// /Chiller_1_Trip
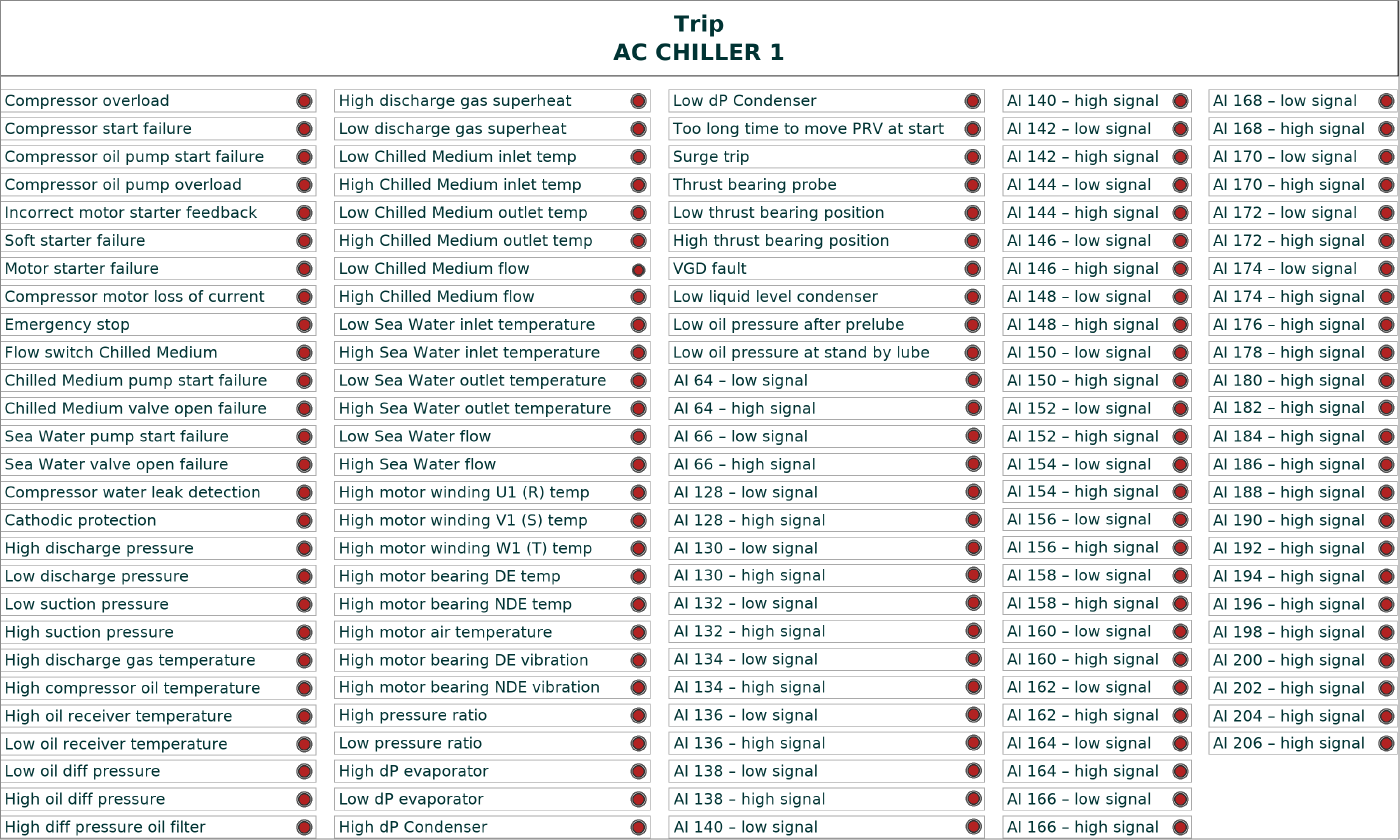
VISUALIZATION Chiller_1_Trip  // 1550x931
    Rectangle (0,0 1548x84)
    Label (318,7 912x70), "Trip AC CHILLER 1"
    Rectangle (0,99 350x25)
    Label (2,101 319x21), "Compressor overload"
    Lamp1 (326,102 22x20), variable: Chiller_1.T_Overload_compressor_motor, style: Lamp-Lamp1-Red
    Rectangle (0,130 350x25)
    Label (2,132 319x21), "Compressor start failure"
    Lamp1 (326,133 22x20), variable: Chiller_1.T_Starter_failure_trip, style: Lamp-Lamp1-Red
    Rectangle (0,161 350x25)
    Label (2,163 319x21), "Compressor oil pump start failure"
    Lamp1 (326,164 22x20), variable: Chiller_1.T_Oil_pump_running_failure, style: Lamp-Lamp1-Red
    Rectangle (0,192 350x25)
    Label (2,194 319x21), "Compressor oil pump overload"
    Lamp1 (326,195 22x20), variable: Chiller_1.T_Overload_oil_pump_motor, style: Lamp-Lamp1-Red
    Rectangle (0,223 350x25)
    Label (2,225 319x21), "Incorrect motor starter feedback"
    Lamp1 (326,226 22x20), variable: Chiller_1.T_Compressor_running_failure, style: Lamp-Lamp1-Red
    Rectangle (0,254 350x25)
    Label (2,256 319x21), "Soft starter failure"
    Lamp1 (326,257 22x20), variable: Chiller_1.T_Softstarter_failure, style: Lamp-Lamp1-Red
    Rectangle (0,285 350x25)
    Label (2,287 319x21), "Motor starter failure"
    Lamp1 (326,288 22x20), variable: Chiller_1.T_Motorstarter_failure, style: Lamp-Lamp1-Red
    Rectangle (0,316 350x25)
    Label (2,318 319x21), "Compressor motor loss of current"
    Lamp1 (326,319 22x20), variable: Chiller_1.T_Comp_motor_power_loss, style: Lamp-Lamp1-Red
    Rectangle (0,347 350x25)
    Label (2,349 319x21), "Emergency stop"
    Lamp1 (326,350 22x20), variable: Chiller_1.T_Emergency_stop, style: Lamp-Lamp1-Red
    Rectangle (0,378 350x25)
    Label (2,380 319x21), "Flow switch Chilled Medium"
    Lamp1 (326,381 22x20), variable: Chiller_1.T_Flow_switch_FT01, style: Lamp-Lamp1-Red
    Rectangle (0,409 350x25)
    Label (2,411 319x21), "Chilled Medium pump start failure"
    Lamp1 (326,412 22x20), variable: Chiller_1.T_Chilled_pump_run_failure, style: Lamp-Lamp1-Red
    Rectangle (0,440 350x25)
    Label (2,442 319x21), "Chilled Medium valve open failure"
    Lamp1 (326,443 22x20), variable: Chiller_1.T_CW_valveopen_failure, style: Lamp-Lamp1-Red
    Rectangle (0,471 350x25)
    Label (2,473 319x21), "Sea Water pump start failure"
    Lamp1 (326,474 22x20), variable: Chiller_1.T_Sea_water_pump_run_failure, style: Lamp-Lamp1-Red
    Rectangle (0,502 350x25)
    Label (2,504 319x21), "Sea Water valve open failure"
    Lamp1 (326,505 22x20), variable: Chiller_1.T_SW_valveopen_failure, style: Lamp-Lamp1-Red
    Rectangle (0,533 350x25)
    Label (2,535 319x21), "Compressor water leak detection"
    Lamp1 (326,536 22x20), variable: Chiller_1.T_Comp_motor_leak_detection, style: Lamp-Lamp1-Red
    Rectangle (0,564 350x25)
    Label (2,566 319x21), "Cathodic protection"
    Lamp1 (326,567 22x20), variable: Chiller_1.T_Cathodic_protect_sys_alarm, style: Lamp-Lamp1-Red
    Rectangle (0,595 350x25)
    Label (2,597 319x21), "High discharge pressure"
    Lamp1 (326,598 22x20), variable: Chiller_1.T_High_discharge_pressure, style: Lamp-Lamp1-Red
    Rectangle (0,626 350x25)
    Label (2,628 319x21), "Low discharge pressure"
    Lamp1 (326,629 22x20), variable: Chiller_1.T_Low_discharge_pressure, style: Lamp-Lamp1-Red
    Rectangle (0,688 350x25)
    Label (2,690 319x21), "High suction pressure"
    Lamp1 (326,691 22x20), variable: Chiller_1.T_High_suction_pressure, style: Lamp-Lamp1-Red
    Rectangle (0,657 350x25)
    Label (2,659 319x21), "Low suction pressure"
    Lamp1 (326,660 22x20), variable: Chiller_1.T_Low_suction_pressure, style: Lamp-Lamp1-Red
    Rectangle (0,719 350x25)
    Label (2,721 319x21), "High discharge gas temperature"
    Lamp1 (326,722 22x20), variable: Chiller_1.T_High_discharge_temp, style: Lamp-Lamp1-Red
    Rectangle (0,750 350x25)
    Label (2,752 319x21), "High compressor oil temperature"
    Lamp1 (326,753 22x20), variable: Chiller_1.T_High_temp_oil_inlet_comp, style: Lamp-Lamp1-Red
    Rectangle (0,781 350x25)
    Label (2,783 319x21), "High oil receiver temperature"
    Lamp1 (326,784 22x20), variable: Chiller_1.T_High_temp_oil_receiver, style: Lamp-Lamp1-Red
    Rectangle (370,749 350x25)
    Label (372,751 319x21), "High motor bearing NDE vibration"
    Lamp1 (696,752 22x20), variable: Chiller_1.T_High_comp_mot_NDE_bear_vib, style: Lamp-Lamp1-Red
    Rectangle (370,780 350x25)
    Label (372,782 319x21), "High pressure ratio"
    Lamp1 (696,783 22x20), variable: Chiller_1.T_High_press_ratio, style: Lamp-Lamp1-Red
    Rectangle (370,811 350x25)
    Label (372,813 319x21), "Low pressure ratio"
    Lamp1 (696,814 22x20), variable: Chiller_1.T_Low_press_ratio, style: Lamp-Lamp1-Red
    Rectangle (370,842 350x25)
    Label (372,844 319x21), "High dP evaporator"
    Lamp1 (696,845 22x20), variable: Chiller_1.T_High_CW_dP, style: Lamp-Lamp1-Red
    Rectangle (370,873 350x25)
    Label (372,875 319x21), "Low dP evaporator"
    Lamp1 (696,876 22x20), variable: Chiller_1.T_Low_CW_dP, style: Lamp-Lamp1-Red
    Rectangle (370,904 350x25)
    Label (372,906 319x21), "High dP Condenser"
    Lamp1 (696,907 22x20), variable: Chiller_1.T_High_SW_dP, style: Lamp-Lamp1-Red
    Rectangle (0,842 350x25)
    Label (2,844 319x21), "Low oil diff pressure"
    Lamp1 (326,845 22x20), variable: Chiller_1.T_Low_oil_diff_pressure, style: Lamp-Lamp1-Red
    Rectangle (0,873 350x25)
    Label (2,875 319x21), "High oil diff pressure"
    Lamp1 (326,876 22x20), variable: Chiller_1.T_High_diff_oil_pressure, style: Lamp-Lamp1-Red
    Rectangle (0,904 350x25)
    Label (2,906 319x21), "High diff pressure oil filter"
    Lamp1 (326,907 22x20), variable: Chiller_1.T_High_oil_filter_diff_press, style: Lamp-Lamp1-Red
    Rectangle (0,812 350x25)
    Label (2,814 319x21), "Low oil receiver temperature"
    Lamp1 (326,815 22x20), variable: Chiller_1.T_Low_temp_oil_receiver, style: Lamp-Lamp1-Red
    Rectangle (370,99 350x25)
    Label (372,101 319x21), "High discharge gas superheat"
    Lamp1 (696,102 22x20), variable: Chiller_1.T_High_disch_superheat, style: Lamp-Lamp1-Red
    Rectangle (370,130 350x25)
    Label (372,132 319x21), "Low discharge gas superheat"
    Lamp1 (696,133 22x20), variable: Chiller_1.T_Low_disch_superheat, style: Lamp-Lamp1-Red
    Rectangle (370,161 350x25)
    Label (372,163 319x21), "Low Chilled Medium inlet temp"
    Lamp1 (696,164 22x20), variable: Chiller_1.T_Low_CW_inlet_temp, style: Lamp-Lamp1-Red
    Rectangle (370,192 350x25)
    Label (372,194 319x21), "High Chilled Medium inlet temp"
    Lamp1 (696,195 22x20), variable: Chiller_1.T_High_CW_inlet_temp, style: Lamp-Lamp1-Red
    Rectangle (370,502 350x25)
    Label (372,504 319x21), "High Sea Water flow"
    Lamp1 (696,505 22x20), variable: Chiller_1.T_High_condenser_flow, style: Lamp-Lamp1-Red
    Rectangle (370,533 350x25)
    Label (372,535 319x21), "High motor winding U1 (R) temp"
    Lamp1 (696,536 22x20), variable: Chiller_1.T_High_motor_wind_temp_R, style: Lamp-Lamp1-Red
    Rectangle (370,564 350x25)
    Label (372,566 319x21), "High motor winding V1 (S) temp"
    Lamp1 (696,567 22x20), variable: Chiller_1.T_High_motor_wind_temp_S, style: Lamp-Lamp1-Red
    Rectangle (370,595 350x25)
    Label (372,597 319x21), "High motor winding W1 (T) temp"
    Lamp1 (696,598 22x20), variable: Chiller_1.T_High_motor_wind_temp_T, style: Lamp-Lamp1-Red
    Rectangle (370,626 350x25)
    Label (372,628 319x21), "High motor bearing DE temp"
    Lamp1 (696,629 22x20), variable: Chiller_1.T_High_comp_mot_DE_bear_temp, style: Lamp-Lamp1-Red
    Rectangle (370,657 350x25)
    Label (372,659 319x21), "High motor bearing NDE temp"
    Lamp1 (696,660 22x20), variable: Chiller_1.T_High_comp_mot_NDE_bear_temp, style: Lamp-Lamp1-Red
    Rectangle (370,688 350x25)
    Label (372,690 319x21), "High motor air temperature"
    Lamp1 (696,691 22x20), variable: Chiller_1.T_High_motor_air_temp, style: Lamp-Lamp1-Red
    Rectangle (370,223 350x25)
    Label (372,225 319x21), "Low Chilled Medium outlet temp"
    Lamp1 (696,226 22x20), variable: Chiller_1.T_Low_CW_outlet_temp, style: Lamp-Lamp1-Red
    Rectangle (370,254 350x25)
    Label (372,256 319x21), "High Chilled Medium outlet temp"
    Lamp1 (696,257 22x20), variable: Chiller_1.T_High_CW_outlet_temp, style: Lamp-Lamp1-Red
    Rectangle (370,285 350x25)
    Label (372,287 330x21), "Low Chilled Medium flow"
    Lamp1 (696,291 22x17), variable: Chiller_1.T_Low_chilled_medium_flow, style: Lamp-Lamp1-Red
    Rectangle (370,347 350x25)
    Label (372,349 319x21), "Low Sea Water inlet temperature"
    Lamp1 (696,350 22x20), variable: Chiller_1.T_Low_SW_inlet_temp, style: Lamp-Lamp1-Red
    Rectangle (370,378 350x25)
    Label (372,380 319x21), "High Sea Water inlet temperature"
    Lamp1 (696,381 22x20), variable: Chiller_1.T_High_SW_inlet_temp, style: Lamp-Lamp1-Red
    Rectangle (370,409 350x25)
    Label (372,411 319x21), "Low Sea Water outlet temperature"
    Lamp1 (696,412 22x20), variable: Chiller_1.T_Low_SW_outlet_temp, style: Lamp-Lamp1-Red
    Rectangle (370,440 350x25)
    Label (372,442 319x21), "High Sea Water outlet temperature"
    Lamp1 (696,443 22x20), variable: Chiller_1.T_High_SW_outlet_temp, style: Lamp-Lamp1-Red
    Rectangle (370,471 350x25)
    Label (372,473 319x21), "Low Sea Water flow"
    Lamp1 (696,474 22x20), variable: Chiller_1.T_Low_condenser_flow, style: Lamp-Lamp1-Red
    Rectangle (370,316 350x25)
    Label (372,318 319x21), "High Chilled Medium flow"
    Lamp1 (696,319 22x20), variable: Chiller_1.T_High_chilled_medium_flow, style: Lamp-Lamp1-Red
    Rectangle (370,719 350x25)
    Label (372,721 319x21), "High motor bearing DE vibration"
    Lamp1 (696,722 22x20), variable: Chiller_1.T_High_comp_mot_DE_bear_vib, style: Lamp-Lamp1-Red
    Rectangle (740,99 350x25)
    Label (742,101 319x21), "Low dP Condenser"
    Lamp1 (1066,102 22x20), variable: Chiller_1.T_Low_SW_dP, style: Lamp-Lamp1-Red
    Rectangle (740,130 350x25)
    Label (742,132 319x21), "Too long time to move PRV at start"
    Lamp1 (1066,133 22x20), variable: Chiller_1.T_Long_time_PRV, style: Lamp-Lamp1-Red
    Rectangle (740,161 350x25)
    Label (742,163 319x21), "Surge trip"
    Lamp1 (1066,164 22x20), variable: Chiller_1.T_Surge_detection, style: Lamp-Lamp1-Red
    Rectangle (740,378 350x25)
    Label (742,380 319x21), "Low oil pressure at stand by lube"
    Lamp1 (1066,381 22x20), variable: Chiller_1.T_Low_oilpress_standby, style: Lamp-Lamp1-Red
    Rectangle (740,192 350x25)
    Label (742,194 319x21), "Thrust bearing probe"
    Lamp1 (1066,195 22x20), variable: Chiller_1.T_Comp_thrust_bearing_position, style: Lamp-Lamp1-Red
    Rectangle (740,223 350x25)
    Label (742,225 319x21), "Low thrust bearing position"
    Lamp1 (1066,226 22x20), variable: Chiller_1.T_Comp_thrust_neg_move, style: Lamp-Lamp1-Red
    Rectangle (740,254 350x25)
    Label (742,256 319x21), "High thrust bearing position"
    Lamp1 (1066,257 22x20), variable: Chiller_1.T_Comp_thrust_pos_move, style: Lamp-Lamp1-Red
    Rectangle (740,285 350x25)
    Label (742,287 319x21), "VGD fault"
    Lamp1 (1066,288 22x20), variable: Chiller_1.T_VGD_fault, style: Lamp-Lamp1-Red
    Rectangle (740,316 350x25)
    Label (742,318 319x21), "Low liquid level condenser"
    Lamp1 (1066,319 22x20), variable: Chiller_1.T_Low_liquid_level, style: Lamp-Lamp1-Red
    Rectangle (740,347 350x25)
    Label (742,349 319x21), "Low oil pressure after prelube"
    Lamp1 (1066,350 22x20), variable: Chiller_1.T_Low_oilpress_prelube, style: Lamp-Lamp1-Red
    Rectangle (1110,316 209x25)
    Rectangle (1110,99 209x25)
    Rectangle (1110,130 209x25)
    Rectangle (1110,161 209x25)
    Rectangle (1110,192 209x25)
    Rectangle (1110,223 209x25)
    Rectangle (1110,254 209x25)
    Rectangle (1110,285 209x25)
    Rectangle (1110,347 209x25)
    Rectangle (1110,378 209x25)
    Rectangle (1110,409 209x25)
    Rectangle (1110,440 209x25)
    Rectangle (1110,471 209x25)
    Rectangle (1110,502 209x25)
    Lamp1 (1296,319 22x20), variable: Chiller_1.T_Sensor_low_signal_AI_148, style: Lamp-Lamp1-Red
    Lamp1 (1296,102 22x20), variable: Chiller_1.T_Sensor_high_signal_AI_140, style: Lamp-Lamp1-Red
    Lamp1 (1296,133 22x20), variable: Chiller_1.T_Sensor_low_signal_AI_142, style: Lamp-Lamp1-Red
    Lamp1 (1296,164 22x20), variable: Chiller_1.T_Sensor_high_signal_AI_142, style: Lamp-Lamp1-Red
    Lamp1 (1296,195 22x20), variable: Chiller_1.T_Sensor_low_signal_AI_144, style: Lamp-Lamp1-Red
    Lamp1 (1296,226 22x20), variable: Chiller_1.T_Sensor_high_signal_AI_144, style: Lamp-Lamp1-Red
    Lamp1 (1296,257 22x20), variable: Chiller_1.T_Sensor_low_signal_AI_146, style: Lamp-Lamp1-Red
    Lamp1 (1296,288 22x20), variable: Chiller_1.T_Sensor_high_signal_AI_146, style: Lamp-Lamp1-Red
    Lamp1 (1296,350 22x20), variable: Chiller_1.T_Sensor_high_signal_AI_148, style: Lamp-Lamp1-Red
    Lamp1 (1296,381 22x20), variable: Chiller_1.T_Sensor_low_signal_AI_150, style: Lamp-Lamp1-Red
    Lamp1 (1296,412 22x20), variable: Chiller_1.T_Sensor_high_signal_AI_150, style: Lamp-Lamp1-Red
    Lamp1 (1296,443 22x20), variable: Chiller_1.T_Sensor_low_signal_AI_152, style: Lamp-Lamp1-Red
    Lamp1 (1296,474 22x20), variable: Chiller_1.T_Sensor_high_signal_AI_152, style: Lamp-Lamp1-Red
    Label (1112,318 179x21), "AI 148 – low signal"
    Label (1112,101 179x21), "AI 140 – high signal"
    Label (1112,132 179x21), "AI 142 – low signal"
    Label (1112,163 179x21), "AI 142 – high signal"
    Label (1112,194 179x21), "AI 144 – low signal"
    Label (1112,225 179x21), "AI 144 – high signal"
    Label (1112,256 179x21), "AI 146 – low signal"
    Label (1112,287 179x21), "AI 146 – high signal"
    Label (1112,349 179x21), "AI 148 – high signal"
    Label (1112,380 179x21), "AI 150 – low signal"
    Label (1112,411 179x21), "AI 150 – high signal"
    Label (1112,442 179x21), "AI 152 – low signal"
    Label (1112,473 179x21), "AI 152 – high signal"
    Label (1112,504 179x21), "AI 154 – low signal"
    Lamp1 (1296,505 22x20), variable: Chiller_1.T_Sensor_low_signal_AI_154, style: Lamp-Lamp1-Red
    Rectangle (1110,532 209x25)
    Label (1112,534 179x21), "AI 154 – high signal"
    Lamp1 (1296,535 22x20), variable: Chiller_1.T_Sensor_high_signal_AI_154, style: Lamp-Lamp1-Red
    Rectangle (1110,563 209x25)
    Rectangle (1110,594 209x25)
    Rectangle (1110,625 209x25)
    Rectangle (1110,656 209x25)
    Rectangle (1110,687 209x25)
    Rectangle (1110,718 209x25)
    Rectangle (1110,749 209x25)
    Rectangle (1110,780 209x25)
    Rectangle (1110,811 209x25)
    Rectangle (1110,842 209x25)
    Rectangle (1110,873 209x25)
    Rectangle (1110,904 209x25)
    Lamp1 (1296,566 22x20), variable: Chiller_1.T_Sensor_low_signal_AI_156, style: Lamp-Lamp1-Red
    Lamp1 (1296,597 22x20), variable: Chiller_1.T_Sensor_high_signal_AI_156, style: Lamp-Lamp1-Red
    Lamp1 (1296,628 22x20), variable: Chiller_1.T_Sensor_low_signal_AI_158, style: Lamp-Lamp1-Red
    Lamp1 (1296,659 22x20), variable: Chiller_1.T_Sensor_high_signal_AI_158, style: Lamp-Lamp1-Red
    Lamp1 (1296,690 22x20), variable: Chiller_1.T_Sensor_low_signal_AI_160, style: Lamp-Lamp1-Red
    Lamp1 (1296,721 22x20), variable: Chiller_1.T_Sensor_high_signal_AI_160, style: Lamp-Lamp1-Red
    Lamp1 (1296,752 22x20), variable: Chiller_1.T_Sensor_low_signal_AI_162, style: Lamp-Lamp1-Red
    Lamp1 (1296,783 22x20), variable: Chiller_1.T_Sensor_high_signal_AI_162, style: Lamp-Lamp1-Red
    Lamp1 (1296,814 22x20), variable: Chiller_1.T_Sensor_low_signal_AI_164, style: Lamp-Lamp1-Red
    Lamp1 (1296,845 22x20), variable: Chiller_1.T_Sensor_high_signal_AI_164, style: Lamp-Lamp1-Red
    Lamp1 (1296,876 22x20), variable: Chiller_1.T_Sensor_low_signal_AI_166, style: Lamp-Lamp1-Red
    Lamp1 (1296,907 22x20), variable: Chiller_1.T_Sensor_high_signal_AI_166, style: Lamp-Lamp1-Red
    Label (1112,565 179x21), "AI 156 – low signal"
    Label (1112,596 179x21), "AI 156 – high signal"
    Label (1112,627 179x21), "AI 158 – low signal"
    Label (1112,658 179x21), "AI 158 – high signal"
    Label (1112,689 179x21), "AI 160 – low signal"
    Label (1112,720 179x21), "AI 160 – high signal"
    Label (1112,751 179x21), "AI 162 – low signal"
    Label (1112,782 179x21), "AI 162 – high signal"
    Label (1112,813 179x21), "AI 164 – low signal"
    Label (1112,844 179x21), "AI 164 – high signal"
    Label (1112,875 179x21), "AI 166 – low signal"
    Label (1112,906 179x21), "AI 166 – high signal"
    Rectangle (1338,223 209x25)
    Rectangle (1338,99 209x25)
    Rectangle (1338,130 209x25)
    Rectangle (1338,161 209x25)
    Rectangle (1338,192 209x25)
    Rectangle (1338,254 209x25)
    Rectangle (1338,285 209x25)
    Rectangle (1338,316 209x25)
    Rectangle (1338,347 209x25)
    Rectangle (1338,378 209x25)
    Rectangle (1338,409 209x25)
    Lamp1 (1524,226 22x20), variable: Chiller_1.T_Sensor_low_signal_AI_172, style: Lamp-Lamp1-Red
    Lamp1 (1524,102 22x20), variable: Chiller_1.T_Sensor_low_signal_AI_168, style: Lamp-Lamp1-Red
    Lamp1 (1524,133 22x20), variable: Chiller_1.T_Sensor_high_signal_AI_168, style: Lamp-Lamp1-Red
    Lamp1 (1524,164 22x20), variable: Chiller_1.T_Sensor_low_signal_AI_170, style: Lamp-Lamp1-Red
    Lamp1 (1524,195 22x20), variable: Chiller_1.T_Sensor_high_signal_AI_170, style: Lamp-Lamp1-Red
    Lamp1 (1524,257 22x20), variable: Chiller_1.T_Sensor_high_signal_AI_172, style: Lamp-Lamp1-Red
    Lamp1 (1524,288 22x20), variable: Chiller_1.T_Sensor_low_signal_AI_174, style: Lamp-Lamp1-Red
    Lamp1 (1524,319 22x20), variable: Chiller_1.T_Sensor_high_signal_AI_174, style: Lamp-Lamp1-Red
    Lamp1 (1524,350 22x20), variable: Chiller_1.T_Sensor_high_signal_AI_176, style: Lamp-Lamp1-Red
    Lamp1 (1524,381 22x20), variable: Chiller_1.T_Sensor_high_signal_AI_178, style: Lamp-Lamp1-Red
    Label (1340,225 179x21), "AI 172 – low signal"
    Label (1340,101 179x21), "AI 168 – low signal"
    Label (1340,132 179x21), "AI 168 – high signal"
    Label (1340,163 179x21), "AI 170 – low signal"
    Label (1340,194 179x21), "AI 170 – high signal"
    Label (1340,256 179x21), "AI 172 – high signal"
    Label (1340,287 179x21), "AI 174 – low signal"
    Label (1340,318 179x21), "AI 174 – high signal"
    Label (1340,349 179x21), "AI 176 – high signal"
    Label (1340,380 179x21), "AI 178 – high signal"
    Label (1340,411 179x21), "AI 180 – high signal"
    Lamp1 (1524,412 22x20), variable: Chiller_1.T_Sensor_high_signal_AI_180, style: Lamp-Lamp1-Red
    Rectangle (1338,439 209x25)
    Label (1340,441 179x21), "AI 182 – high signal"
    Lamp1 (1524,442 22x20), variable: Chiller_1.T_Sensor_high_signal_AI_182, style: Lamp-Lamp1-Red
    Rectangle (740,656 350x25)
    Rectangle (740,687 350x25)
    Rectangle (740,718 350x25)
    Rectangle (740,749 350x25)
    Rectangle (740,780 350x25)
    Rectangle (740,811 350x25)
    Rectangle (740,842 350x25)
    Rectangle (740,873 350x25)
    Rectangle (740,904 350x25)
    Label (743,658 299x21), "AI 132 – low signal"
    Label (743,689 299x21), "AI 132 – high signal"
    Label (743,720 299x21), "AI 134 – low signal"
    Label (743,751 299x21), "AI 134 – high signal"
    Label (743,782 299x21), "AI 136 – low signal"
    Label (743,813 299x21), "AI 136 – high signal"
    Label (743,844 299x21), "AI 138 – low signal"
    Label (743,875 299x21), "AI 138 – high signal"
    Label (743,906 299x21), "AI 140 – low signal"
    Rectangle (740,625 350x25)
    Rectangle (740,502 350x25)
    Rectangle (740,533 350x25)
    Rectangle (740,564 350x25)
    Rectangle (740,595 350x25)
    Rectangle (740,409 350x25)
    Rectangle (740,440 350x25)
    Rectangle (740,471 350x25)
    Label (743,504 298x21), "AI 66 – high signal"
    Label (743,535 298x21), "AI 128 – low signal"
    Label (743,566 298x21), "AI 128 – high signal"
    Label (743,597 298x21), "AI 130 – low signal"
    Label (743,411 298x21), "AI 64 – low signal"
    Label (743,442 298x21), "AI 64 – high signal"
    Label (743,473 298x21), "AI 66 – low signal"
    Label (743,627 350x21), "AI 130 – high signal"
    Lamp1 (1066,658 24x20), variable: Chiller_1.T_Sensor_low_signal_AI_132, style: Lamp-Lamp1-Red
    Lamp1 (1066,689 24x20), variable: Chiller_1.T_Sensor_high_signal_AI_132, style: Lamp-Lamp1-Red
    Lamp1 (1066,720 24x20), variable: Chiller_1.T_Sensor_low_signal_AI_134, style: Lamp-Lamp1-Red
    Lamp1 (1066,751 24x20), variable: Chiller_1.T_Sensor_high_signal_AI_134, style: Lamp-Lamp1-Red
    Lamp1 (1066,782 24x20), variable: Chiller_1.T_Sensor_low_signal_AI_136, style: Lamp-Lamp1-Red
    Lamp1 (1066,813 24x20), variable: Chiller_1.T_Sensor_high_signal_AI_136, style: Lamp-Lamp1-Red
    Lamp1 (1066,844 24x20), variable: Chiller_1.T_Sensor_low_signal_AI_138, style: Lamp-Lamp1-Red
    Lamp1 (1066,875 24x20), variable: Chiller_1.T_Sensor_high_signal_AI_138, style: Lamp-Lamp1-Red
    Lamp1 (1066,906 24x20), variable: Chiller_1.T_Sensor_low_signal_AI_140, style: Lamp-Lamp1-Red
    Lamp1 (1066,504 24x20), variable: Chiller_1.T_Sensor_high_signal_AI_66, style: Lamp-Lamp1-Red
    Lamp1 (1066,535 24x20), variable: Chiller_1.T_Sensor_low_signal_AI_128, style: Lamp-Lamp1-Red
    Lamp1 (1066,566 24x20), variable: Chiller_1.T_Sensor_high_signal_AI_128, style: Lamp-Lamp1-Red
    Lamp1 (1066,597 24x20), variable: Chiller_1.T_Sensor_low_signal_AI_130, style: Lamp-Lamp1-Red
    Lamp1 (1066,411 24x20), variable: Chiller_1.T_Sensor_low_signal_AI_64, style: Lamp-Lamp1-Red
    Lamp1 (1066,442 24x20), variable: Chiller_1.T_Sensor_high_signal_AI_64, style: Lamp-Lamp1-Red
    Lamp1 (1066,473 24x20), variable: Chiller_1.T_Sensor_low_signal_AI_66, style: Lamp-Lamp1-Red
    Lamp1 (1066,627 24x20), variable: Chiller_1.T_Sensor_high_signal_AI_130, style: Lamp-Lamp1-Red
    Rectangle (1338,595 209x25)
    Rectangle (1338,471 209x25)
    Rectangle (1338,502 209x25)
    Rectangle (1338,533 209x25)
    Rectangle (1338,564 209x25)
    Rectangle (1338,626 209x25)
    Rectangle (1338,657 209x25)
    Rectangle (1338,688 209x25)
    Rectangle (1338,719 209x25)
    Rectangle (1338,750 209x25)
    Rectangle (1338,781 209x25)
    Lamp1 (1524,598 22x20), variable: Chiller_1.T_Sensor_high_signal_AI_192, style: Lamp-Lamp1-Red
    Lamp1 (1524,474 22x20), variable: Chiller_1.T_Sensor_high_signal_AI_184, style: Lamp-Lamp1-Red
    Lamp1 (1524,505 22x20), variable: Chiller_1.T_Sensor_high_signal_AI_186, style: Lamp-Lamp1-Red
    Lamp1 (1524,536 22x20), variable: Chiller_1.T_Sensor_high_signal_AI_188, style: Lamp-Lamp1-Red
    Lamp1 (1524,567 22x20), variable: Chiller_1.T_Sensor_high_signal_AI_190, style: Lamp-Lamp1-Red
    Lamp1 (1524,629 22x20), variable: Chiller_1.T_Sensor_high_signal_AI_194, style: Lamp-Lamp1-Red
    Lamp1 (1524,660 22x20), variable: Chiller_1.T_Sensor_high_signal_AI_196, style: Lamp-Lamp1-Red
    Lamp1 (1524,691 22x20), variable: Chiller_1.T_Sensor_high_signal_AI_198, style: Lamp-Lamp1-Red
    Lamp1 (1524,722 22x20), variable: Chiller_1.T_Sensor_high_signal_AI_200, style: Lamp-Lamp1-Red
    Lamp1 (1524,753 22x20), variable: Chiller_1.T_Sensor_high_signal_AI_202, style: Lamp-Lamp1-Red
    Label (1340,597 179x21), "AI 192 – high signal"
    Label (1340,473 179x21), "AI 184 – high signal"
    Label (1340,504 179x21), "AI 186 – high signal"
    Label (1340,535 179x21), "AI 188 – high signal"
    Label (1340,566 179x21), "AI 190 – high signal"
    Label (1340,628 179x21), "AI 194 – high signal"
    Label (1340,659 179x21), "AI 196 – high signal"
    Label (1340,690 179x21), "AI 198 – high signal"
    Label (1340,721 179x21), "AI 200 – high signal"
    Label (1340,752 179x21), "AI 202 – high signal"
    Label (1340,783 179x21), "AI 204 – high signal"
    Lamp1 (1524,784 22x20), variable: Chiller_1.T_Sensor_high_signal_AI_204, style: Lamp-Lamp1-Red
    Rectangle (1338,811 209x25)
    Label (1340,813 179x21), "AI 206 – high signal"
    Lamp1 (1524,814 22x20), variable: Chiller_1.T_Sensor_high_signal_AI_206, style: Lamp-Lamp1-Red
END_VISUALIZATION

// /Chiller_1_Values
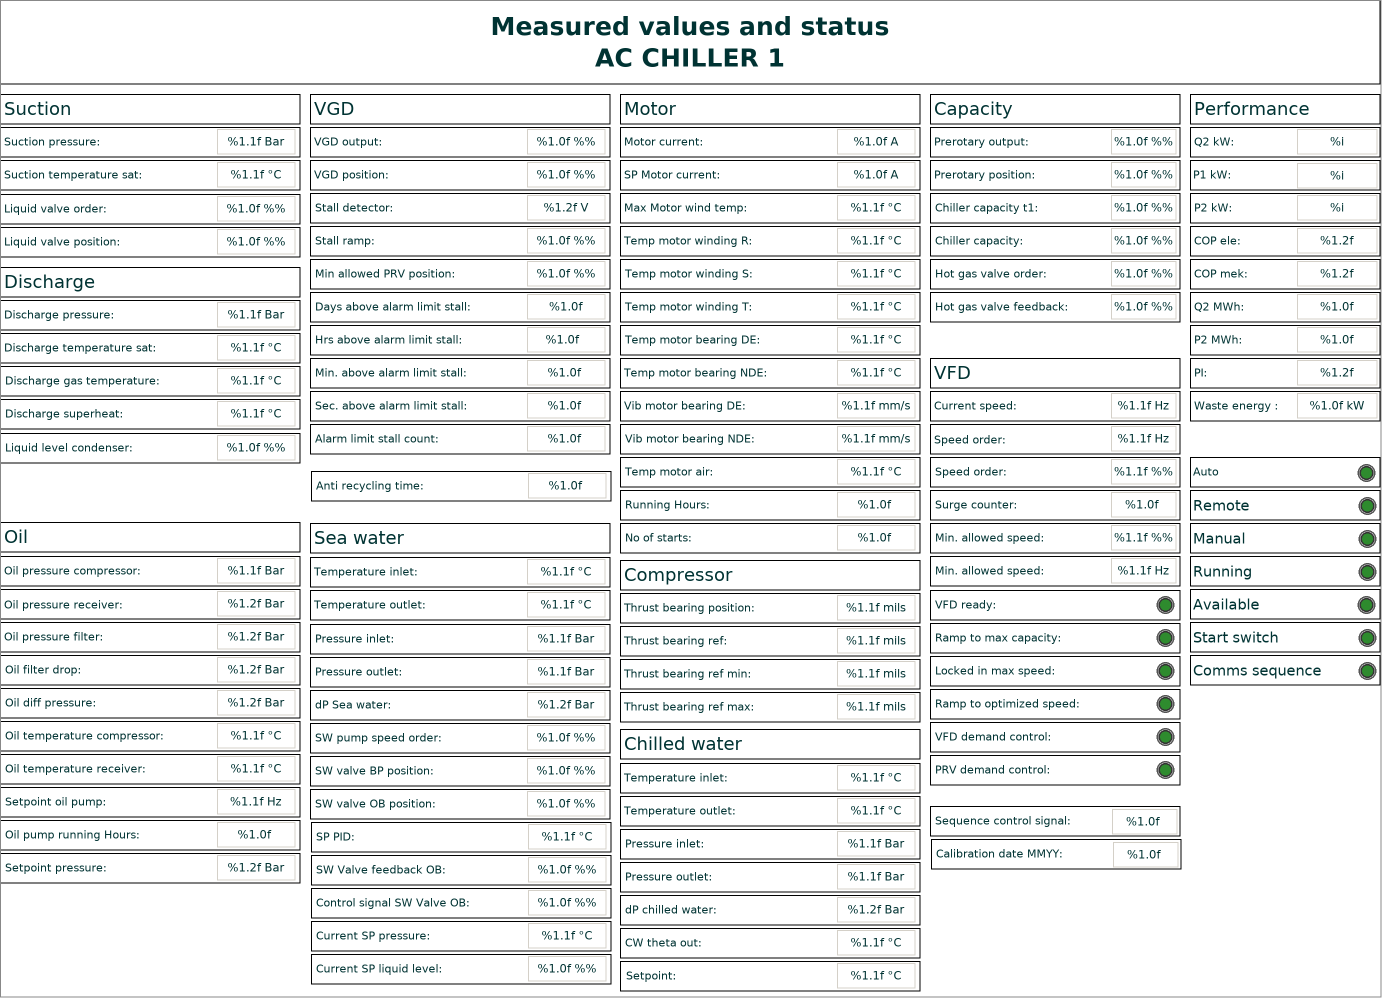
VISUALIZATION Chiller_1_Values  // 1382x998
    Rectangle (0,0 1380x84)
    Label (234,7 912x70), "Measured values and status AC CHILLER 1"
    Rectangle (0,94 300x30)
    Label (1,94 215x30), "Suction"
    Rectangle (0,127 300x30)
    Label (1,122 208x40), "Suction pressure:"
    Textfield (217,129 78x25), "%1.1f Bar", tooltip "Chiller_1.Press_suction_compr", text variable: Chiller_1.Press_suction_compr
        p4168582468: Chiller_1.Press_suction_compr
    Rectangle (0,160 300x30)
    Label (1,155 209x40), "Suction temperature sat:"
    Textfield (217,162 78x25), "%1.1f °C", tooltip "Chiller_1.Suction_saturated_temp", text variable: Chiller_1.Suction_saturated_temp
        p4168582468: Chiller_1.Suction_saturated_temp
    Rectangle (0,194 300x30)
    Label (1,189 211x40), "Liquid valve order:"
    Textfield (217,196 78x25), "%1.0f %%", tooltip "Chiller_1.Liquid_valve_output", text variable: Chiller_1.Liquid_valve_output
        p4168582468: Chiller_1.Liquid_valve_output
    Rectangle (0,227 300x30)
    Label (1,222 216x40), "Liquid valve position:"
    Textfield (217,229 78x25), "%1.0f %%", tooltip "Chiller_1.Feedback_liquid_valve", text variable: Chiller_1.Feedback_liquid_valve
        p4168582468: Chiller_1.Feedback_liquid_valve
    Rectangle (0,267 300x30)
    Label (1,267 194x30), "Discharge"
    Rectangle (0,300 300x30)
    Label (1,295 213x40), "Discharge pressure:"
    Textfield (217,302 78x25), "%1.1f Bar", tooltip "Chiller_1.Press_discharge_compr", text variable: Chiller_1.Press_discharge_compr
        p4168582468: Chiller_1.Press_discharge_compr
    Rectangle (0,333 300x30)
    Label (1,328 214x40), "Discharge temperature sat:"
    Textfield (217,335 78x25), "%1.1f °C", tooltip "Chiller_1.Discharge_saturated_temp", text variable: Chiller_1.Discharge_saturated_temp
        p4168582468: Chiller_1.Discharge_saturated_temp
    Rectangle (0,366 300x30)
    Label (2,361 213x40), "Discharge gas temperature:"
    Textfield (217,368 78x25), "%1.1f °C", tooltip "Chiller_1.Temp_discharge", text variable: Chiller_1.Temp_discharge
        p4168582468: Chiller_1.Temp_discharge
    Rectangle (0,433 300x30)
    Textfield (217,435 78x25), "%1.0f %%", tooltip "Chiller_1.Liquid_level_condenser", text variable: Chiller_1.Liquid_level_condenser
        p4168582468: Chiller_1.Liquid_level_condenser
    Rectangle (0,399 300x30)
    Label (2,394 212x40), "Discharge superheat:"
    Textfield (217,401 78x25), "%1.1f °C", tooltip "Chiller_1.Discharge_superheat", text variable: Chiller_1.Discharge_superheat
        p4168582468: Chiller_1.Discharge_superheat
    Rectangle (620,729 300x30)
    Label (621,729 194x30), "Chilled water"
    Rectangle (620,763 300x30)
    Label (621,758 204x40), "Temperature inlet:"
    Textfield (837,765 78x25), "%1.1f °C", tooltip "Chiller_1.Temp_chilled_medium_in", text variable: Chiller_1.Temp_chilled_medium_in
        p4168582468: Chiller_1.Temp_chilled_medium_in
    Rectangle (620,796 300x30)
    Label (621,791 209x40), "Temperature outlet:"
    Textfield (837,798 78x25), "%1.1f °C", tooltip "Chiller_1.Temp_chilled_medium_out", text variable: Chiller_1.Temp_chilled_medium_out
        p4168582468: Chiller_1.Temp_chilled_medium_out
    Rectangle (620,829 300x30)
    Label (622,824 206x40), "Pressure inlet:"
    Textfield (837,831 78x25), "%1.1f Bar", tooltip "Chiller_1.Press_chilled_medium_in", text variable: Chiller_1.Press_chilled_medium_in
        p4168582468: Chiller_1.Press_chilled_medium_in
    Rectangle (620,862 300x30)
    Label (622,857 208x40), "Pressure outlet:"
    Textfield (837,864 78x25), "%1.1f Bar", tooltip "Chiller_1.Press_chilled_medium_out", text variable: Chiller_1.Press_chilled_medium_out
        p4168582468: Chiller_1.Press_chilled_medium_out
    Rectangle (620,895 300x30)
    Label (622,890 207x40), "dP chilled water:"
    Textfield (837,897 78x25), "%1.2f Bar", tooltip "Chiller_1.dP_CW", text variable: Chiller_1.dP_CW
        p4168582468: Chiller_1.dP_CW
    Rectangle (620,928 300x30)
    Label (622,923 205x40), "CW theta out:"
    Textfield (837,930 78x25), "%1.1f °C", tooltip "Chiller_1.Theta_out", text variable: Chiller_1.Theta_out
        p4168582468: Chiller_1.Theta_out
    Rectangle (310,94 300x30)
    Label (311,94 194x30), "VGD"
    Rectangle (310,127 300x30)
    Label (311,122 209x40), "VGD output:"
    Textfield (527,129 78x25), "%1.0f %%", tooltip "Chiller_1.VGD_output", text variable: Chiller_1.VGD_output
        p4168582468: Chiller_1.VGD_output
    Rectangle (310,160 300x30)
    Label (311,155 204x40), "VGD position:"
    Textfield (527,162 78x25), "%1.0f %%", tooltip "Chiller_1.Feedback_VGD", text variable: Chiller_1.Feedback_VGD
        p4168582468: Chiller_1.Feedback_VGD
    Rectangle (310,193 300x30)
    Label (312,188 209x40), "Stall detector:"
    Textfield (527,195 78x25), "%1.2f V", tooltip "Chiller_1.Stall_detector", text variable: Chiller_1.Stall_detector
        p4168582468: Chiller_1.Stall_detector
    Rectangle (310,226 300x30)
    Label (312,221 178x40), "Stall ramp:"
    Textfield (527,228 78x25), "%1.0f %%", tooltip "Chiller_1.Stall_ramp", text variable: Chiller_1.Stall_ramp
        p4168582468: Chiller_1.Stall_ramp
    Rectangle (310,259 300x30)
    Label (312,254 216x40), "Min allowed PRV position:"
    Textfield (527,261 78x25), "%1.0f %%", tooltip "Chiller_1.Min_allowed_PRVposition", text variable: Chiller_1.Min_allowed_PRVposition
        p4168582468: Chiller_1.Min_allowed_PRVposition
    Rectangle (310,292 300x30)
    Label (312,287 216x40), "Days above alarm limit stall:"
    Textfield (527,294 78x25), "%1.0f", tooltip "Chiller_1.Days_above_stall_limit", text variable: Chiller_1.Days_above_stall_limit
        p4168582468: Chiller_1.Days_above_stall_limit
    Rectangle (310,325 300x30)
    Label (312,320 215x40), "Hrs above alarm limit stall:"
    Textfield (527,327 78x25), "%1.0f", tooltip "Chiller_1.Hrs_above_stall_limit", text variable: Chiller_1.Hrs_above_stall_limit
        p4168582468: Chiller_1.Hrs_above_stall_limit
    Rectangle (310,358 300x30)
    Label (312,353 218x40), "Min. above alarm limit stall:"
    Textfield (527,360 78x25), "%1.0f", tooltip "Chiller_1.Min_above_stall_limit", text variable: Chiller_1.Min_above_stall_limit
        p4168582468: Chiller_1.Min_above_stall_limit
    Rectangle (310,391 300x30)
    Label (312,386 214x40), "Sec. above alarm limit stall:"
    Textfield (527,393 78x25), "%1.0f", tooltip "Chiller_1.Sec_above_stall_limit", text variable: Chiller_1.Sec_above_stall_limit
        p4168582468: Chiller_1.Sec_above_stall_limit
    Rectangle (310,424 300x30)
    Label (312,419 216x40), "Alarm limit stall count:"
    Textfield (527,426 78x25), "%1.0f", tooltip "Chiller_1.Alarm_limit_stall_count", text variable: Chiller_1.Alarm_limit_stall_count
        p4168582468: Chiller_1.Alarm_limit_stall_count
    Rectangle (930,94 250x30)
    Label (931,94 162x30), "Capacity"
    Rectangle (930,127 250x30)
    Label (931,126 174x32), "Prerotary output:"
    Textfield (1111,129 65x25), "%1.0f %%", tooltip "Chiller_1.Prerotary_output", text variable: Chiller_1.Prerotary_output
        p4168582468: Chiller_1.Prerotary_output
    Rectangle (930,160 250x30)
    Label (931,159 173x32), "Prerotary position:"
    Textfield (1111,162 65x25), "%1.0f %%", tooltip "Chiller_1.Feedback_PRV", text variable: Chiller_1.Feedback_PRV
        p4168582468: Chiller_1.Feedback_PRV
    Rectangle (930,259 250x30)
    Label (932,258 177x32), "Hot gas valve order:"
    Textfield (1111,261 65x25), "%1.0f %%", tooltip "Chiller_1.Hot_gas_valve_output", text variable: Chiller_1.Hot_gas_valve_output
        p4168582468: Chiller_1.Hot_gas_valve_output
    Rectangle (930,292 250x30)
    Label (932,293 177x28), "Hot gas valve feedback:"
    Textfield (1111,294 65x25), "%1.0f %%", tooltip "Chiller_1.Feedback_HGV", text variable: Chiller_1.Feedback_HGV
        p4168582468: Chiller_1.Feedback_HGV
    Label (2,428 210x40), "Liquid level condenser:"
    Rectangle (310,523 300x30)
    Label (311,523 194x30), "Sea water"
    Rectangle (310,557 300x30)
    Label (311,552 211x40), "Temperature inlet:"
    Textfield (527,559 78x25), "%1.1f °C", tooltip "Chiller_1.Temp_water_inlet_cond", text variable: Chiller_1.Temp_water_inlet_cond
        p4168582468: Chiller_1.Temp_water_inlet_cond
    Rectangle (310,624 300x30)
    Label (312,619 210x40), "Pressure inlet:"
    Textfield (527,626 78x25), "%1.1f Bar", tooltip "Chiller_1.Press_water_cond_inlet", text variable: Chiller_1.Press_water_cond_inlet
        p4168582468: Chiller_1.Press_water_cond_inlet
    Rectangle (310,657 300x30)
    Label (312,652 210x40), "Pressure outlet:"
    Textfield (527,659 78x25), "%1.1f Bar", tooltip "Chiller_1.Press_water_cond_out", text variable: Chiller_1.Press_water_cond_out
        p4168582468: Chiller_1.Press_water_cond_out
    Rectangle (310,690 300x30)
    Label (312,685 210x40), "dP Sea water:"
    Textfield (527,692 78x25), "%1.2f Bar", tooltip "Chiller_1.dP_CW", text variable: Chiller_1.dP_SW
        p4168582468: Chiller_1.dP_SW
    Rectangle (310,723 300x30)
    Label (312,718 216x40), "SW pump speed order:"
    Textfield (527,725 78x25), "%1.0f %%", tooltip "Chiller_1.SW_pump_speed_order", text variable: Chiller_1.SW_pump_speed_order
        p4168582468: Chiller_1.SW_pump_speed_order
    Rectangle (310,756 300x30)
    Label (312,751 212x40), "SW valve BP position:"
    Textfield (527,758 78x25), "%1.0f %%", tooltip "Chiller_1.Order_SWW_bypass", text variable: Chiller_1.Order_SWW_bypass
        p4168582468: Chiller_1.Order_SWW_bypass
    Rectangle (310,789 300x30)
    Label (312,784 208x40), "SW valve OB position:"
    Textfield (527,791 78x25), "%1.0f %%", tooltip "Chiller_1.Order_SWW_overboard", text variable: Chiller_1.Order_SWW_overboard
        p4168582468: Chiller_1.Order_SWW_overboard
    Rectangle (310,590 300x30)
    Label (311,585 211x40), "Temperature outlet:"
    Textfield (527,592 78x25), "%1.1f °C", tooltip "Chiller_1.Temp_water_outlet_cond", text variable: Chiller_1.Temp_water_outlet_cond
        p4168582468: Chiller_1.Temp_water_outlet_cond
    Rectangle (0,522 300x30)
    Label (1,522 194x30), "Oil"
    Rectangle (0,556 300x30)
    Label (1,551 211x40), "Oil pressure compressor:"
    Textfield (217,558 78x25), "%1.1f Bar", tooltip "Chiller_1.Press_oil_compr", text variable: Chiller_1.Press_oil_compr
        p4168582468: Chiller_1.Press_oil_compr
    Rectangle (0,589 300x30)
    Label (1,585 210x40), "Oil pressure receiver:"
    Textfield (217,591 78x25), "%1.2f Bar", tooltip "Chiller_1.Press_oil_receiver", text variable: Chiller_1.Press_oil_receiver
        p4168582468: Chiller_1.Press_oil_receiver
    Rectangle (0,655 300x30)
    Label (2,650 209x40), "Oil filter drop:"
    Textfield (217,657 78x25), "%1.2f Bar", tooltip "Chiller_1.Oil_Filter_Drop", text variable: Chiller_1.Oil_Filter_Drop
        p4168582468: Chiller_1.Oil_Filter_Drop
    Rectangle (0,721 300x30)
    Label (2,716 218x40), "Oil temperature compressor:"
    Textfield (217,723 78x25), "%1.1f °C", tooltip "Chiller_1.Temp_oil_inlet_compr", text variable: Chiller_1.Temp_oil_inlet_compr
        p4168582468: Chiller_1.Temp_oil_inlet_compr
    Rectangle (0,754 300x30)
    Label (2,749 210x40), "Oil temperature receiver:"
    Textfield (217,756 78x25), "%1.1f °C", tooltip "Chiller_1.Oil_temp_receiver", text variable: Chiller_1.Oil_temp_receiver
        p4168582468: Chiller_1.Oil_temp_receiver
    Rectangle (0,688 300x30)
    Label (2,683 211x40), "Oil diff pressure:"
    Textfield (217,690 78x25), "%1.2f Bar", tooltip "Chiller_1.Oil_diff_pressure", text variable: Chiller_1.Oil_diff_pressure
        p4168582468: Chiller_1.Oil_diff_pressure
    Rectangle (0,787 300x30)
    Label (2,782 212x40), "Setpoint oil pump:"
    Textfield (217,789 78x25), "%1.1f Hz", tooltip "Chiller_1.Setpoint_conv_oil_pump", text variable: Chiller_1.Setpoint_conv_oil_pump
        p4168582468: Chiller_1.Setpoint_conv_oil_pump
    Rectangle (0,820 300x30)
    Label (2,815 206x40), "Oil pump running Hours:"
    Textfield (217,822 78x25), "%1.0f", tooltip "Chiller_1.Oil_pump_running_hours", text variable: Chiller_1.Oil_pump_running_hours
        p4168582468: Chiller_1.Oil_pump_running_hours
    Rectangle (0,622 300x30)
    Label (1,617 210x40), "Oil pressure filter:"
    Textfield (217,624 78x25), "%1.2f Bar", tooltip "Chiller_1.Oil_pressure_before_filter", text variable: Chiller_1.Oil_pressure_before_filter
        p4168582468: Chiller_1.Oil_pressure_before_filter
    Rectangle (620,560 300x30)
    Label (621,560 194x30), "Compressor"
    Rectangle (620,593 300x30)
    Label (621,592 216x32), "Thrust bearing position:"
    Textfield (837,595 78x25), "%1.1f mils", tooltip "Chiller_1.Thrust_bearing_position", text variable: Chiller_1.Thrust_bearing_position
        p4168582468: Chiller_1.Thrust_bearing_position
    Rectangle (620,659 300x30)
    Label (621,658 208x32), "Thrust bearing ref min:"
    Textfield (837,661 78x25), "%1.1f mils", tooltip "Chiller_1.Thrust_bearing_ref_min", text variable: Chiller_1.Thrust_bearing_ref_min
        p4168582468: Chiller_1.Thrust_bearing_ref_min
    Rectangle (1190,226 190x30)
    Label (1191,228 112x26), "COP ele:"
    Textfield (1297,228 80x25), "%1.2f", tooltip "Chiller_1.COP_chiller_ele", text variable: Chiller_1.COP_chiller_ele
        p4168582468: Chiller_1.COP_chiller_ele
    Rectangle (1190,94 190x30)
    Label (1191,94 123x30), "Performance"
    Rectangle (1190,127 190x30)
    Label (1191,126 112x32), "Q2 kW:"
    Textfield (1297,129 80x25), "%i", tooltip "Chiller_1.Chiller_capacity_kW", text variable: Chiller_1.Chiller_capacity_kW
        p4168582468: Chiller_1.Chiller_capacity_kW
    Rectangle (1190,193 190x30)
    Label (1191,194 112x28), "P2 kW:"
    Textfield (1297,195 80x25), "%i", tooltip "Chiller_1.P2_mot_1_kW", text variable: Chiller_1.P2_mot_1_kW
        p4168582468: Chiller_1.P2_mot_1_kW
    Rectangle (1190,160 190x30)
    Textfield (1297,163 80x25), "%i", tooltip "Chiller_1.P1_motor_kW", text variable: Chiller_1.P1_motor_kW
        p4168582468: Chiller_1.P1_motor_kW
    Label (1190,159 112x32), "P1 kW:"
    Rectangle (1190,457 190x30)
    Lamp1 (1355,463 23x20), tooltip "Chiller_1.Unit_auto", variable: Chiller_1.Unit_auto, style: Lamp-Lamp1-Green
    Label (1190,459 112x26), "Auto"
    Rectangle (1190,490 190x30)
    Rectangle (1190,523 190x30)
    Rectangle (1190,556 190x30)
    Rectangle (1190,589 190x30)
    Rectangle (1190,622 190x30)
    Rectangle (1190,655 190x30)
    Label (1190,495 105x21), "Remote"
    Lamp1 (1356,496 23x20), tooltip "Chiller_1.Unit_remote", variable: Chiller_1.Unit_remote, style: Lamp-Lamp1-Green
    Label (1190,528 105x21), "Manual"
    Lamp1 (1356,529 23x20), tooltip "Chiller_1.Unit_manual", variable: Chiller_1.Unit_manual, style: Lamp-Lamp1-Green
    Label (1190,561 105x21), "Running"
    Lamp1 (1356,562 23x20), tooltip "Chiller_1.Unit_running", variable: Chiller_1.Unit_running, style: Lamp-Lamp1-Green
    Label (1190,594 105x21), "Available"
    Lamp1 (1355,595 23x20), tooltip "Chiller_1.Unit_avabiable", variable: Chiller_1.Unit_available, style: Lamp-Lamp1-Green
    Label (1190,627 130x21), "Start switch"
    Lamp1 (1356,628 23x20), tooltip "Chiller_1.Unit_start_switch", variable: Chiller_1.Unit_start_switch, style: Lamp-Lamp1-Green
    Lamp1 (1356,661 23x20), tooltip "Sequence.A_Comms_chiller_1", variable: not.Sequence.A_Comms_chiller_1, style: Lamp-Lamp1-Green
    Label (1190,660 148x21), "Comms sequence"
    Rectangle (1190,292 190x30)
    Label (1191,293 112x28), "Q2 MWh:"
    Textfield (1297,294 80x25), "%1.0f", tooltip "Chiller_1.Q2_chillerMWh", text variable: Chiller_1.Q2_chillerMWh
        p4168582468: Chiller_1.Q2_chillerMWh
    Rectangle (930,358 250x30)
    Label (931,358 162x30), "VFD"
    Rectangle (930,391 250x30)
    Label (931,390 173x32), "Current speed:"
    Textfield (1111,393 65x25), "%1.1f Hz", tooltip "Chiller_1.Speed_feedback_VFD", text variable: Chiller_1.Speed_feedback_VFD
        p4168582468: Chiller_1.Speed_feedback_VFD
    Rectangle (930,424 250x30)
    Label (931,420 167x40), "Speed order:"
    Textfield (1111,426 65x25), "%1.1f Hz", tooltip "Chiller_1.Order_VFD_Hz", text variable: Chiller_1.Order_VFD_Hz
        p4168582468: Chiller_1.Order_VFD_Hz
    Rectangle (930,457 250x30)
    Label (932,455 171x34), "Speed order:"
    Textfield (1111,459 65x25), "%1.1f %%", tooltip "Chiller_1.Order_VFD_perc", text variable: Chiller_1.Order_VFD_perc
        p4168582468: Chiller_1.Order_VFD_perc
    Rectangle (930,490 250x30)
    Label (932,492 170x26), "Surge counter:"
    Textfield (1111,492 65x25), "%1.0f", tooltip "Chiller_1.Surge_counter_VFD", text variable: Chiller_1.Surge_counter_VFD
        p4168582468: Chiller_1.Surge_counter_VFD
    Rectangle (930,523 250x30)
    Label (932,522 176x32), "Min. allowed speed:"
    Textfield (1111,525 65x25), "%1.1f %%", tooltip "Chiller_1.Opt_speed_VFD_perc", text variable: Chiller_1.Opt_speed_VFD_perc
        p4168582468: Chiller_1.Opt_speed_VFD_perc
    Rectangle (930,556 250x30)
    Label (932,554 177x34), "Min. allowed speed:"
    Textfield (1111,558 65x25), "%1.1f Hz", tooltip "Chiller_1.Opt_speed_VFD_Hz", text variable: Chiller_1.Opt_speed_VFD_Hz
        p4168582468: Chiller_1.Opt_speed_VFD_Hz
    Rectangle (930,193 250x30)
    Label (932,192 174x32), "Chiller capacity t1:"
    Textfield (1111,195 65x25), "%1.0f %%", tooltip "Chiller_1.Chiller_capacity_t1", text variable: Chiller_1.Chiller_capacity_t1
        p4168582468: Chiller_1.Chiller_capacity_t1
    Rectangle (620,94 300x30)
    Label (621,94 194x30), "Motor"
    Rectangle (620,127 300x30)
    Label (621,122 209x40), "Motor current:"
    Textfield (837,129 78x25), "%1.0f A", tooltip "Chiller_1.Motor_current", text variable: Chiller_1.Motor_current
        p4168582468: Chiller_1.Motor_current
    Rectangle (620,226 300x30)
    Label (621,221 210x40), "Temp motor winding R:"
    Textfield (837,228 78x25), "%1.1f °C", tooltip "Chiller_1.Temp_motor_wind_R", text variable: Chiller_1.Temp_motor_wind_R
        p4168582468: Chiller_1.Temp_motor_wind_R
    Rectangle (620,259 300x30)
    Label (622,254 204x40), "Temp motor winding S:"
    Textfield (837,261 78x25), "%1.1f °C", tooltip "Chiller_1.Temp_motor_wind_S", text variable: Chiller_1.Temp_motor_wind_S
        p4168582468: Chiller_1.Temp_motor_wind_S
    Rectangle (620,292 300x30)
    Label (622,287 206x40), "Temp motor winding T:"
    Textfield (837,294 78x25), "%1.1f °C", tooltip "Chiller_1.Temp_motor_wind_T", text variable: Chiller_1.Temp_motor_wind_T
        p4168582468: Chiller_1.Temp_motor_wind_T
    Rectangle (620,325 300x30)
    Label (622,320 216x40), "Temp motor bearing DE:"
    Textfield (837,327 78x25), "%1.1f °C", tooltip "Chiller_1.Temp_motor_bearing_DE", text variable: Chiller_1.Temp_motor_bearing_DE
        p4168582468: Chiller_1.Temp_motor_bearing_DE
    Rectangle (620,358 300x30)
    Label (621,353 218x40), "Temp motor bearing NDE:"
    Textfield (837,360 78x25), "%1.1f °C", tooltip "Chiller_1.Temp_motor_bearing_NDE", text variable: Chiller_1.Temp_motor_bearing_NDE
        p4168582468: Chiller_1.Temp_motor_bearing_NDE
    Rectangle (620,391 300x30)
    Label (621,386 215x40), "Vib motor bearing DE:"
    Textfield (837,393 78x25), "%1.1f mm/s", tooltip "Chiller_1.Vibration_compressor_DE", text variable: Chiller_1.Vibration_compressor_DE
        p4168582468: Chiller_1.Vibration_compressor_DE
    Rectangle (620,424 300x30)
    Label (622,419 215x40), "Vib motor bearing NDE:"
    Textfield (837,426 78x25), "%1.1f mm/s", tooltip "Chiller_1.Vibration_compressor_NDE", text variable: Chiller_1.Vibration_compressor_NDE
        p4168582468: Chiller_1.Vibration_compressor_NDE
    Rectangle (620,457 300x30)
    Label (622,452 210x40), "Temp motor air:"
    Textfield (837,459 78x25), "%1.1f °C", tooltip "Chiller_1.Temp_motor_air", text variable: Chiller_1.Temp_motor_air
        p4168582468: Chiller_1.Temp_motor_air
    Rectangle (620,490 300x30)
    Label (622,485 204x40), "Running Hours:"
    Textfield (837,492 78x25), "%1.0f", tooltip "Chiller_1.Running_hours_compressormotor", text variable: Chiller_1.Running_hours_compressormotor
        p4168582468: Chiller_1.Running_hours_compressormotor
    Rectangle (620,523 300x30)
    Label (622,518 207x40), "No of starts:"
    Textfield (837,525 78x25), "%1.0f", tooltip "Chiller_1.Number_of_starts", text variable: Chiller_1.Number_of_starts
        p4168582468: Chiller_1.Number_of_starts
    Rectangle (930,590 250x30)
    Label (932,588 177x34), "VFD ready:"
    Lamp1 (1154,595 23x20), tooltip "Chiller_1.VFD_ready", variable: Chiller_1.VFD_ready, style: Lamp-Lamp1-Green
    Rectangle (930,623 250x30)
    Label (932,621 209x34), "Ramp to max capacity:"
    Lamp1 (1154,628 23x20), tooltip "Chiller_1.VFD_ramp_100_perc", variable: Chiller_1.VFD_ramp_100_perc, style: Lamp-Lamp1-Green
    Rectangle (930,656 250x30)
    Label (932,654 209x34), "Locked in max speed:"
    Lamp1 (1154,661 23x20), tooltip "Chiller_1.VFD_locked_100_perc", variable: Chiller_1.VFD_locked_100_perc, style: Lamp-Lamp1-Green
    Rectangle (930,689 250x30)
    Label (932,687 209x34), "Ramp to optimized speed:"
    Lamp1 (1154,694 23x20), tooltip "Chiller_1.VFD_ramp_d_PRVcontrol", variable: Chiller_1.VFD_ramp_d_PRVcontrol, style: Lamp-Lamp1-Green
    Rectangle (930,722 250x30)
    Label (932,720 209x34), "VFD demand control:"
    Lamp1 (1154,727 23x20), tooltip "Chiller_1.VFD_control", variable: Chiller_1.VFD_control, style: Lamp-Lamp1-Green
    Rectangle (930,755 250x30)
    Label (932,753 209x34), "PRV demand control:"
    Lamp1 (1154,760 23x20), tooltip "Chiller_1.PRV_control", variable: Chiller_1.PRV_control, style: Lamp-Lamp1-Green
    Rectangle (620,961 300x30)
    Label (623,956 205x40), "Setpoint:"
    Textfield (837,963 78x25), "%1.1f °C", tooltip "Chiller_1.SP_CW_controller", text variable: Chiller_1.SP_CW_controller
        p4168582468: Chiller_1.SP_CW_controller
    Rectangle (311,822 300x30)
    Label (313,817 208x40), "SP PID:"
    Textfield (528,824 78x25), "%1.1f °C", tooltip "Chiller_1.SP_PID_seawater", text variable: Chiller_1.SP_PID_seawater
        p4168582468: Chiller_1.SP_PID_seawater
    Rectangle (1190,259 190x30)
    Label (1191,261 112x26), "COP mek:"
    Textfield (1297,261 80x25), "%1.2f", tooltip "Chiller_1.COP_chiller_mech", text variable: Chiller_1.COP_chiller_mech
        p4168582468: Chiller_1.COP_chiller_mech
    Rectangle (620,692 300x30)
    Label (621,691 208x32), "Thrust bearing ref max:"
    Textfield (837,694 78x25), "%1.1f mils", tooltip "Chiller_1.Thrust_bearing_ref_max", text variable: Chiller_1.Thrust_bearing_ref_max
        p4168582468: Chiller_1.Thrust_bearing_ref_max
    Rectangle (620,160 300x30)
    Label (621,155 209x40), "SP Motor current:"
    Textfield (837,162 78x25), "%1.0f A", tooltip "Chiller_1.SP_MC_controller", text variable: Chiller_1.SP_MC_controller
        p4168582468: Chiller_1.SP_MC_controller
    Rectangle (620,626 300x30)
    Label (621,625 216x32), "Thrust bearing ref:"
    Textfield (837,628 78x25), "%1.1f mils", tooltip "Chiller_1.Thrust_bearing_ref", text variable: Chiller_1.Thrust_bearing_ref
        p4168582468: Chiller_1.Thrust_bearing_ref
    Rectangle (311,471 300x30)
    Label (313,466 216x40), "Anti recycling time:"
    Textfield (528,473 78x25), "%1.0f", tooltip "Chiller_1.Anti_recycle_time", text variable: Chiller_1.Anti_recycle_time
        p4168582468: Chiller_1.Anti_recycle_time
    Rectangle (0,853 300x30)
    Label (2,848 211x40), "Setpoint pressure:"
    Textfield (217,855 78x25), "%1.2f Bar", tooltip "Chiller_1.SP_oil_pressure", text variable: Chiller_1.SP_oil_pressure
        p4168582468: Chiller_1.SP_oil_pressure
    Rectangle (311,855 300x30)
    Label (313,850 208x40), "SW Valve feedback OB:"
    Textfield (528,857 78x25), "%1.0f %%", tooltip "Chiller_1.Feedback_seawater_valve_overboard", text variable: Chiller_1.Feedback_seawater_valve_overboard
        p4168582468: Chiller_1.Feedback_seawater_valve_overboard
    Rectangle (620,193 300x30)
    Label (621,188 210x40), "Max Motor wind temp:"
    Textfield (837,195 78x25), "%1.1f °C", tooltip "Chiller_1.Max_motor_wind_temp", text variable: Chiller_1.Max_motor_wind_temp
        p4168582468: Chiller_1.Max_motor_wind_temp
    Rectangle (311,888 300x30)
    Label (313,883 208x40), "Control signal SW Valve OB:"
    Textfield (528,890 78x25), "%1.0f %%", tooltip "Chiller_1.Feedback_seawater_valve_overboard", text variable: Chiller_1.Feedback_seawater_valve_overboard
        p4168582468: Chiller_1.Feedback_seawater_valve_overboard
    Rectangle (311,921 300x30)
    Label (313,916 208x40), "Current SP pressure:"
    Textfield (528,923 78x25), "%1.1f °C", tooltip "Chiller_1.SP_PID_seawater", text variable: Chiller_1.SP_cond_press
        p4168582468: Chiller_1.SP_PID_seawater
    Rectangle (311,954 300x30)
    Label (313,949 208x40), "Current SP liquid level:"
    Textfield (528,956 78x25), "%1.0f %%", tooltip "Chiller_1.SP_PID_Level", text variable: Chiller_1.SP_PID_Level
        p4168582468: Chiller_1.SP_PID_Level
    Rectangle (930,806 250x30)
    Label (932,804 183x34), "Sequence control signal:"
    Rectangle (1190,358 190x30)
    Label (1191,360 112x26), "PI:"
    Textfield (1297,360 80x25), "%1.2f", tooltip "Chiller_1.PI_chiller", text variable: Chiller_1.PI_chiller
        p4168582468: Chiller_1.PI_chiller
    Rectangle (1190,391 190x30)
    Label (1191,393 112x26), "Waste energy :"
    Textfield (1297,393 80x25), "%1.0f kW", tooltip "Chiller_1.Wasted_energy_kW", text variable: Chiller_1.Wasted_energy_kW
        p4168582468: Chiller_1.Wasted_energy_kW
    Rectangle (1190,325 190x30)
    Label (1191,327 112x26), "P2 MWh:"
    Textfield (1297,327 80x25), "%1.0f", tooltip "Chiller_1.Chiller_P2_MWh", text variable: Chiller_1.Chiller_P2_MWh
        p4168582468: Chiller_1.Chiller_P2_MWh
    Textfield (1112,809 65x25), "%1.0f", tooltip "Chiller_1.Control_signal_unit_d", text variable: Chiller_1.Control_signal_unit_d
        p4168582468: Chiller_1.Control_signal_unit_d
    Rectangle (931,839 250x30)
    Label (933,837 183x34), "Calibration date MMYY:"
    Textfield (1113,842 65x25), "%1.0f", tooltip "Chiller_1.Cal_date_MMYY", text variable: Chiller_1.Cal_date_MMYY
        p4168582468: Chiller_1.Cal_date_MMYY
    Rectangle (930,226 250x30)
    Label (932,225 174x32), "Chiller capacity:"
    Textfield (1111,228 65x25), "%1.0f %%", tooltip "Chiller_1.Chiller_capacity", text variable: Chiller_1.Chiller_capacity
        p4168582468: Chiller_1.Chiller_capacity
END_VISUALIZATION

// /Chiller_1_VFD
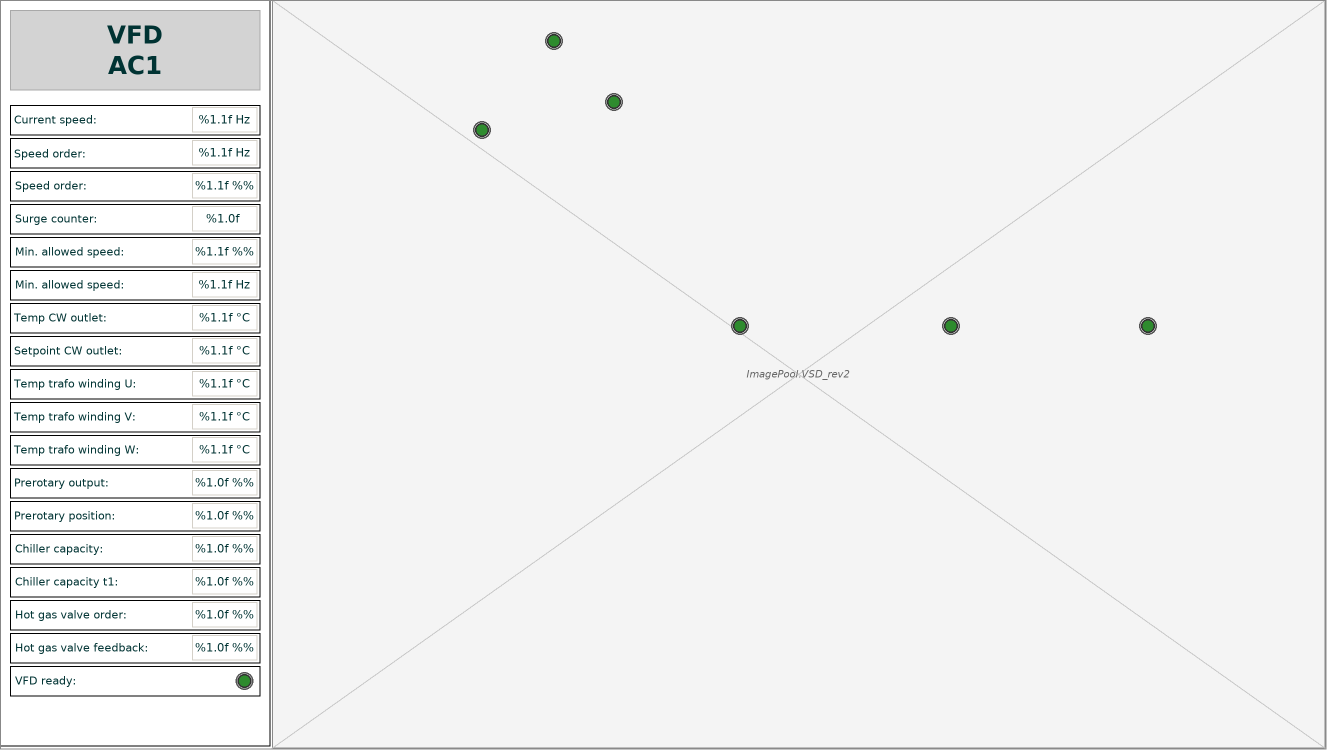
VISUALIZATION Chiller_1_VFD  // 1327x750
    Image (272,0 1053x748), image: ImagePool.VSD_rev2
    Rectangle (0,0 270x746)
    Lamp1 (469,120 26x20), variable: Chiller_1.VFD_ramp_100_perc, style: Lamp-Lamp1-Green
    Lamp1 (541,31 26x20), variable: Chiller_1.VFD_locked_100_perc, style: Lamp-Lamp1-Green
    Lamp1 (601,92 26x20), variable: Chiller_1.VFD_ramp_d_PRVcontrol, style: Lamp-Lamp1-Green
    Lamp1 (727,316 26x20), variable: Chiller_1.PRV_control, style: Lamp-Lamp1-Green
    Lamp1 (938,316 26x20), variable: Chiller_1.VFD_control, style: Lamp-Lamp1-Green
    Lamp1 (1135,316 26x20), variable: Chiller_1.PRV_control, style: Lamp-Lamp1-Green
    Textfield (10,10 250x80), "VFD AC1", text index: Sequence.Seq_cap_order_C3
    Rectangle (10,666 250x30)
    Label (12,664 177x34), "VFD ready:"
    Lamp1 (233,671 23x20), tooltip "Chiller_1.VFD_ready", variable: Chiller_1.VFD_ready, style: Lamp-Lamp1-Green
    Rectangle (10,105 250x30)
    Label (11,104 173x32), "Current speed:"
    Textfield (192,107 65x25), "%1.1f Hz", tooltip "Chiller_1.Speed_feedback_VFD", text variable: Chiller_1.Speed_feedback_VFD
        p4168582468: Chiller_1.Speed_feedback_VFD
    Rectangle (10,138 250x30)
    Label (11,134 167x40), "Speed order:"
    Textfield (192,140 65x25), "%1.1f Hz", tooltip "Chiller_1.Order_VFD_Hz", text variable: Chiller_1.Order_VFD_Hz
        p4168582468: Chiller_1.Order_VFD_Hz
    Rectangle (10,171 250x30)
    Label (12,169 171x34), "Speed order:"
    Textfield (192,173 65x25), "%1.1f %%", tooltip "Chiller_1.Order_VFD_perc", text variable: Chiller_1.Order_VFD_perc
        p4168582468: Chiller_1.Order_VFD_perc
    Rectangle (10,204 250x30)
    Label (12,206 170x26), "Surge counter:"
    Textfield (192,206 65x25), "%1.0f", tooltip "Chiller_1.Surge_counter_VFD", text variable: Chiller_1.Surge_counter_VFD
        p4168582468: Chiller_1.Surge_counter_VFD
    Rectangle (10,237 250x30)
    Label (12,236 176x32), "Min. allowed speed:"
    Textfield (192,239 65x25), "%1.1f %%", tooltip "Chiller_1.Opt_speed_VFD_perc", text variable: Chiller_1.Opt_speed_VFD_perc
        p4168582468: Chiller_1.Opt_speed_VFD_perc
    Rectangle (10,270 250x30)
    Label (12,268 177x34), "Min. allowed speed:"
    Textfield (192,272 65x25), "%1.1f Hz", tooltip "Chiller_1.Opt_speed_VFD_Hz", text variable: Chiller_1.Opt_speed_VFD_Hz
        p4168582468: Chiller_1.Opt_speed_VFD_Hz
    Rectangle (10,303 250x30)
    Label (11,305 169x26), "Temp CW outlet:"
    Textfield (192,305 65x25), "%1.1f °C", tooltip "Chiller_1.Temp_chilled_medium_out", text variable: Chiller_1.Temp_chilled_medium_out
        p4168582468: Chiller_1.Temp_chilled_medium_out
    Rectangle (10,336 250x30)
    Label (11,338 169x26), "Setpoint CW outlet:"
    Textfield (192,338 65x25), "%1.1f °C", tooltip "Chiller_1.SP_CW_controller", text variable: Chiller_1.SP_CW_controller
        p4168582468: Chiller_1.SP_CW_controller
    Rectangle (10,369 250x30)
    Label (11,371 169x26), "Temp trafo winding U:"
    Textfield (192,371 65x25), "%1.1f °C", tooltip "Chiller_1.Temp_motor_wind_R", text variable: Chiller_1.Temp_motor_wind_R
        p4168582468: Chiller_1.Temp_motor_wind_R
    Rectangle (10,402 250x30)
    Label (11,404 169x26), "Temp trafo winding V:"
    Textfield (192,404 65x25), "%1.1f °C", tooltip "Chiller_1.Temp_motor_wind_S", text variable: Chiller_1.Temp_motor_wind_S
        p4168582468: Chiller_1.Temp_motor_wind_S
    Rectangle (10,435 250x30)
    Label (11,437 169x26), "Temp trafo winding W:"
    Textfield (192,437 65x25), "%1.1f °C", tooltip "Chiller_1.Temp_motor_wind_T", text variable: Chiller_1.Temp_motor_wind_T
        p4168582468: Chiller_1.Temp_motor_wind_T
    Rectangle (10,468 250x30)
    Label (11,467 174x32), "Prerotary output:"
    Textfield (192,470 65x25), "%1.0f %%", tooltip "Chiller_1.Prerotary_output", text variable: Chiller_1.Prerotary_output
        p4168582468: Chiller_1.Prerotary_output
    Rectangle (10,501 250x30)
    Label (11,500 173x32), "Prerotary position:"
    Textfield (192,503 65x25), "%1.0f %%", tooltip "Chiller_1.Feedback_PRV", text variable: Chiller_1.Feedback_PRV
        p4168582468: Chiller_1.Feedback_PRV
    Rectangle (10,534 250x30)
    Label (12,533 174x32), "Chiller capacity:"
    Textfield (192,536 65x25), "%1.0f %%", tooltip "Chiller_1.Chiller_capacity", text variable: Chiller_1.Chiller_capacity
        p4168582468: Chiller_1.Chiller_capacity
    Rectangle (10,600 250x30)
    Label (12,599 177x32), "Hot gas valve order:"
    Textfield (192,602 65x25), "%1.0f %%", tooltip "Chiller_1.Hot_gas_valve_output", text variable: Chiller_1.Hot_gas_valve_output
        p4168582468: Chiller_1.Hot_gas_valve_output
    Rectangle (10,633 250x30)
    Label (12,634 177x28), "Hot gas valve feedback:"
    Textfield (192,635 65x25), "%1.0f %%", tooltip "Chiller_1.Feedback_HGV", text variable: Chiller_1.Feedback_HGV
        p4168582468: Chiller_1.Feedback_HGV
    Rectangle (10,567 250x30)
    Label (12,566 174x32), "Chiller capacity t1:"
    Textfield (192,569 65x25), "%1.0f %%", tooltip "Chiller_1.Chiller_capacity_t1", text variable: Chiller_1.Chiller_capacity_t1
        p4168582468: Chiller_1.Chiller_capacity_t1
    Rectangle (432,18 87x711), colour toggle: Chiller_1.VFD_ramp_100_perc
    Rectangle (518,18 65x711), colour toggle: Chiller_1.VFD_locked_100_perc
    Rectangle (583,18 57x711), colour toggle: Chiller_1.VFD_ramp_d_PRVcontrol
    Rectangle (641,18 199x711), colour toggle: Chiller_1.PRV_control
    Rectangle (1066,18 162x711), colour toggle: Chiller_1.PRV_control
    Rectangle (841,18 225x711), colour toggle: Chiller_1.VFD_control
END_VISUALIZATION

// /Chiller_2_Alarm
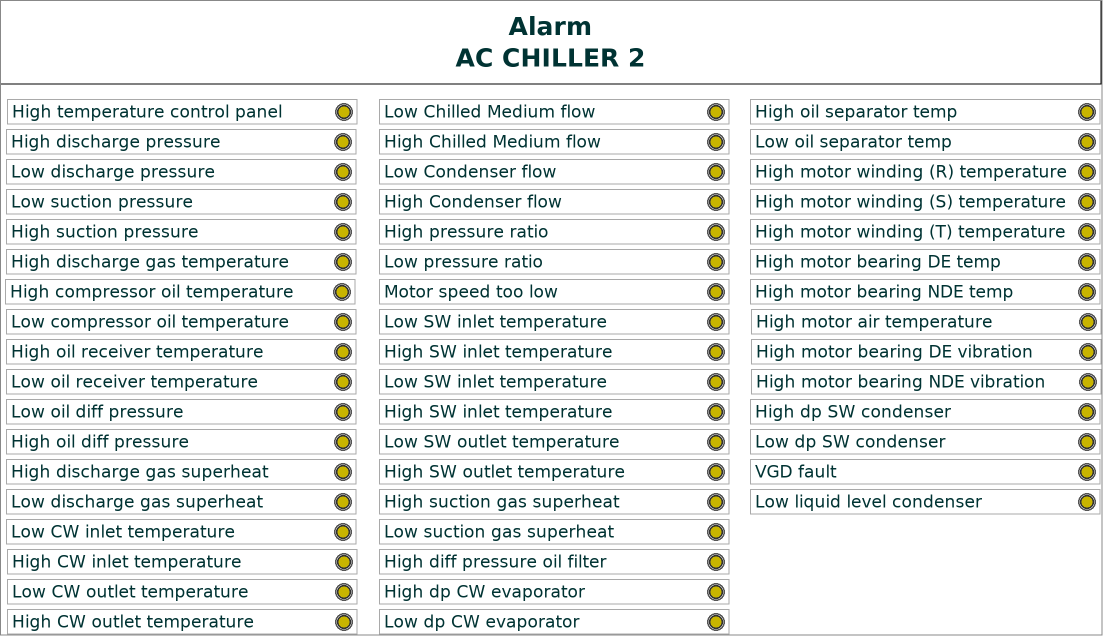
VISUALIZATION Chiller_2_Alarm  // 1103x636
    Rectangle (0,0 1101x84)
    Label (19,7 1063x70), "Alarm AC CHILLER 2"
    Rectangle (6,129 350x25)
    Label (8,131 318x21), "High discharge pressure"
    Lamp1 (332,132 22x20), variable: Chiller_2.A_high_disch_press, style: Lamp-Lamp1-Yellow
    Rectangle (6,189 350x25)
    Label (8,191 319x21), "Low suction pressure"
    Lamp1 (332,192 22x20), variable: Chiller_2.A_Low_suction_pressure, style: Lamp-Lamp1-Yellow
    Rectangle (6,219 350x25)
    Label (8,221 322x21), "High suction pressure"
    Lamp1 (332,222 22x20), variable: Chiller_2.A_High_suction_pressure, style: Lamp-Lamp1-Yellow
    Rectangle (6,249 350x25)
    Label (8,251 317x21), "High discharge gas temperature"
    Lamp1 (332,252 22x20), variable: Chiller_2.A_High_discharge_temp, style: Lamp-Lamp1-Yellow
    Rectangle (750,159 350x25)
    Label (752,161 320x21), "High motor winding (R) temperature"
    Lamp1 (1076,162 22x20), variable: Chiller_2.A_High_motor_wind_temp_R, style: Lamp-Lamp1-Yellow
    Rectangle (750,189 350x25)
    Label (752,191 319x21), "High motor winding (S) temperature"
    Lamp1 (1076,192 22x20), variable: Chiller_2.A_High_motor_wind_temp_S, style: Lamp-Lamp1-Yellow
    Rectangle (6,489 350x25)
    Label (8,491 319x21), "Low discharge gas superheat"
    Lamp1 (332,492 22x20), variable: Chiller_2.A_Low_discharge_superheat, style: Lamp-Lamp1-Yellow
    Rectangle (6,459 350x25)
    Label (8,461 322x21), "High discharge gas superheat"
    Lamp1 (332,462 22x20), variable: Chiller_2.A_High_discharge_superheat, style: Lamp-Lamp1-Yellow
    Rectangle (6,339 350x25)
    Label (8,341 317x21), "High oil receiver temperature"
    Lamp1 (332,342 22x20), variable: Chiller_2.A_High_oil_temp_receiver, style: Lamp-Lamp1-Yellow
    Rectangle (6,369 350x25)
    Label (8,371 319x21), "Low oil receiver temperature"
    Lamp1 (332,372 22x20), variable: Chiller_2.A_Low_oil_temp_receiver, style: Lamp-Lamp1-Yellow
    Rectangle (6,399 350x25)
    Label (8,401 322x21), "Low oil diff pressure"
    Lamp1 (332,402 22x20), variable: Chiller_2.A_Low_oil_diff_pressure, style: Lamp-Lamp1-Yellow
    Rectangle (6,429 350x25)
    Label (8,431 317x21), "High oil diff pressure"
    Lamp1 (332,432 22x20), variable: Chiller_2.A_High_oil_diff_pressure, style: Lamp-Lamp1-Yellow
    Rectangle (6,309 350x25)
    Label (8,311 319x21), "Low compressor oil temperature"
    Lamp1 (332,312 22x20), variable: Chiller_2.A_Low_temp_oil_inlet_comp, style: Lamp-Lamp1-Yellow
    Rectangle (5,279 350x25)
    Label (7,281 322x21), "High compressor oil temperature"
    Lamp1 (331,282 22x20), variable: Chiller_2.A_High_temp_oil_inlet_comp, style: Lamp-Lamp1-Yellow
    Rectangle (379,309 350x25)
    Label (381,311 317x21), "Low SW inlet temperature"
    Lamp1 (705,312 22x20), variable: Chiller_2.A_Low_SW_inlet_temp, style: Lamp-Lamp1-Yellow
    Rectangle (7,549 350x25)
    Label (9,551 322x21), "High CW inlet temperature"
    Lamp1 (333,552 22x20), variable: Chiller_2.A_High_CW_inlet_temp, style: Lamp-Lamp1-Yellow
    Rectangle (6,519 350x25)
    Label (8,521 317x21), "Low CW inlet temperature"
    Lamp1 (332,522 22x20), variable: Chiller_2.A_Low_CW_inlet_temp, style: Lamp-Lamp1-Yellow
    Rectangle (379,549 350x25)
    Label (381,551 317x21), "High diff pressure oil filter"
    Lamp1 (705,552 22x20), variable: Chiller_2.A_High_oil_filter_diff_press, style: Lamp-Lamp1-Yellow
    Rectangle (750,219 350x25)
    Label (752,221 317x21), "High motor winding (T) temperature"
    Lamp1 (1076,222 22x20), variable: Chiller_2.A_High_motor_wind_temp_T, style: Lamp-Lamp1-Yellow
    Rectangle (750,249 350x25)
    Label (752,251 317x21), "High motor bearing DE temp"
    Lamp1 (1076,252 22x20), variable: Chiller_2.A_High_comp_mo_DE_bear_temp, style: Lamp-Lamp1-Yellow
    Rectangle (750,279 350x25)
    Label (752,281 319x21), "High motor bearing NDE temp"
    Lamp1 (1076,282 22x20), variable: Chiller_2.A_High_comp_mo_NDE_bear_temp, style: Lamp-Lamp1-Yellow
    Rectangle (751,309 350x25)
    Label (753,311 322x21), "High motor air temperature"
    Lamp1 (1077,312 22x20), variable: Chiller_2.A_High_motor_air_temp, style: Lamp-Lamp1-Yellow
    Rectangle (751,339 350x25)
    Label (753,341 317x21), "High motor bearing DE vibration"
    Lamp1 (1077,342 22x20), variable: Chiller_2.A_High_comp_mo_DE_bear_vib, style: Lamp-Lamp1-Yellow
    Rectangle (751,369 350x25)
    Label (753,371 319x21), "High motor bearing NDE vibration"
    Lamp1 (1077,372 22x20), variable: Chiller_2.A_High_comp_mo_NDE_bear_vib, style: Lamp-Lamp1-Yellow
    Rectangle (379,579 350x25)
    Label (381,581 322x21), "High dp CW evaporator"
    Lamp1 (705,582 22x20), variable: Chiller_2.A_High_CW_dP, style: Lamp-Lamp1-Yellow
    Rectangle (379,609 350x25)
    Label (381,611 317x21), "Low dp CW evaporator"
    Lamp1 (705,612 22x20), variable: Chiller_2.A_Low_CW_dP, style: Lamp-Lamp1-Yellow
    Rectangle (750,399 350x25)
    Label (752,401 319x21), "High dp SW condenser"
    Lamp1 (1076,402 22x20), variable: Chiller_2.A_High_SW_dP, style: Lamp-Lamp1-Yellow
    Rectangle (750,429 350x25)
    Label (752,431 322x21), "Low dp SW condenser"
    Lamp1 (1076,432 22x20), variable: Chiller_2.A_Low_SW_dP, style: Lamp-Lamp1-Yellow
    Rectangle (750,459 350x25)
    Label (752,461 317x21), "VGD fault"
    Lamp1 (1076,462 22x20), variable: Chiller_2.A_VGD_Fault, style: Lamp-Lamp1-Yellow
    Rectangle (750,489 350x25)
    Label (752,491 317x21), "Low liquid level condenser"
    Lamp1 (1076,492 22x20), variable: Chiller_2.A_Low_liquid_level, style: Lamp-Lamp1-Yellow
    Rectangle (6,159 350x25)
    Label (8,161 318x21), "Low discharge pressure"
    Lamp1 (332,162 22x20), variable: Chiller_2.A_low_disch_press, style: Lamp-Lamp1-Yellow
    Rectangle (379,339 350x25)
    Label (381,341 314x21), "High SW inlet temperature"
    Lamp1 (705,342 22x20), variable: Chiller_2.A_High_SW_inlet_temp, style: Lamp-Lamp1-Yellow
    Rectangle (7,99 350x25)
    Label (9,101 318x21), "High temperature control panel"
    Lamp1 (333,102 22x20), variable: Chiller_2.A_low_disch_press, style: Lamp-Lamp1-Yellow
    Rectangle (7,579 350x25)
    Label (9,581 317x21), "Low CW outlet temperature"
    Lamp1 (333,582 22x20), variable: Chiller_2.A_Low_CW_outlet_temp, style: Lamp-Lamp1-Yellow
    Rectangle (7,609 350x25)
    Label (9,611 317x21), "High CW outlet temperature"
    Lamp1 (333,612 22x20), variable: Chiller_2.A_high_CW_outlet_temp, style: Lamp-Lamp1-Yellow
    Rectangle (379,99 350x25)
    Label (381,101 317x21), "Low Chilled Medium flow"
    Lamp1 (705,102 22x20), variable: Chiller_2.A_Low_chilled_medium_flow, style: Lamp-Lamp1-Yellow
    Rectangle (379,129 350x25)
    Label (381,131 317x21), "High Chilled Medium flow"
    Lamp1 (705,132 22x20), variable: Chiller_2.A_High_chilled_medium_flow, style: Lamp-Lamp1-Yellow
    Rectangle (379,159 350x25)
    Label (381,161 317x21), "Low Condenser flow"
    Lamp1 (705,162 22x20), variable: Chiller_2.A_Low_condenser_flow, style: Lamp-Lamp1-Yellow
    Rectangle (379,189 350x25)
    Label (381,191 317x21), "High Condenser flow"
    Lamp1 (705,192 22x20), variable: Chiller_2.A_High_condenser_flow, style: Lamp-Lamp1-Yellow
    Rectangle (379,219 350x25)
    Label (381,221 317x21), "High pressure ratio"
    Lamp1 (705,222 22x20), variable: Chiller_2.A_High_press_ratio, style: Lamp-Lamp1-Yellow
    Rectangle (379,249 350x25)
    Label (381,251 317x21), "Low pressure ratio"
    Lamp1 (705,252 22x20), variable: Chiller_2.A_Low_press_ratio, style: Lamp-Lamp1-Yellow
    Rectangle (379,279 350x25)
    Label (381,281 317x21), "Motor speed too low"
    Lamp1 (705,282 22x20), variable: Chiller_2.A_Motor_speed_low, style: Lamp-Lamp1-Yellow
    Rectangle (379,369 350x25)
    Label (381,371 317x21), "Low SW inlet temperature"
    Lamp1 (705,372 22x20), variable: Chiller_2.A_Low_SW_inlet_temp, style: Lamp-Lamp1-Yellow
    Rectangle (379,399 350x25)
    Label (381,401 314x21), "High SW inlet temperature"
    Lamp1 (705,402 22x20), variable: Chiller_2.A_High_SW_inlet_temp, style: Lamp-Lamp1-Yellow
    Rectangle (379,429 350x25)
    Label (381,431 317x21), "Low SW outlet temperature"
    Lamp1 (705,432 22x20), variable: Chiller_2.A_Low_SW_outlet_temp, style: Lamp-Lamp1-Yellow
    Rectangle (379,459 350x25)
    Label (381,461 314x21), "High SW outlet temperature"
    Lamp1 (705,462 22x20), variable: Chiller_2.A_High_SW_outlet_temp, style: Lamp-Lamp1-Yellow
    Rectangle (379,489 350x25)
    Label (381,491 317x21), "High suction gas superheat"
    Lamp1 (705,492 22x20), variable: Chiller_2.A_High_suction_superheat, style: Lamp-Lamp1-Yellow
    Rectangle (379,519 350x25)
    Label (381,521 314x21), "Low suction gas superheat"
    Lamp1 (705,522 22x20), variable: Chiller_2.A_Low_suction_superheat, style: Lamp-Lamp1-Yellow
    Rectangle (750,99 350x25)
    Label (752,101 317x21), "High oil separator temp"
    Lamp1 (1076,102 22x20), variable: Chiller_2.A_High_temp_oil_separator, style: Lamp-Lamp1-Yellow
    Rectangle (750,129 350x25)
    Label (752,131 319x21), "Low oil separator temp"
    Lamp1 (1076,132 22x20), variable: Chiller_2.A_Low_temp_oil_separator, style: Lamp-Lamp1-Yellow
END_VISUALIZATION

// /Chiller_2_Flow_Diagram
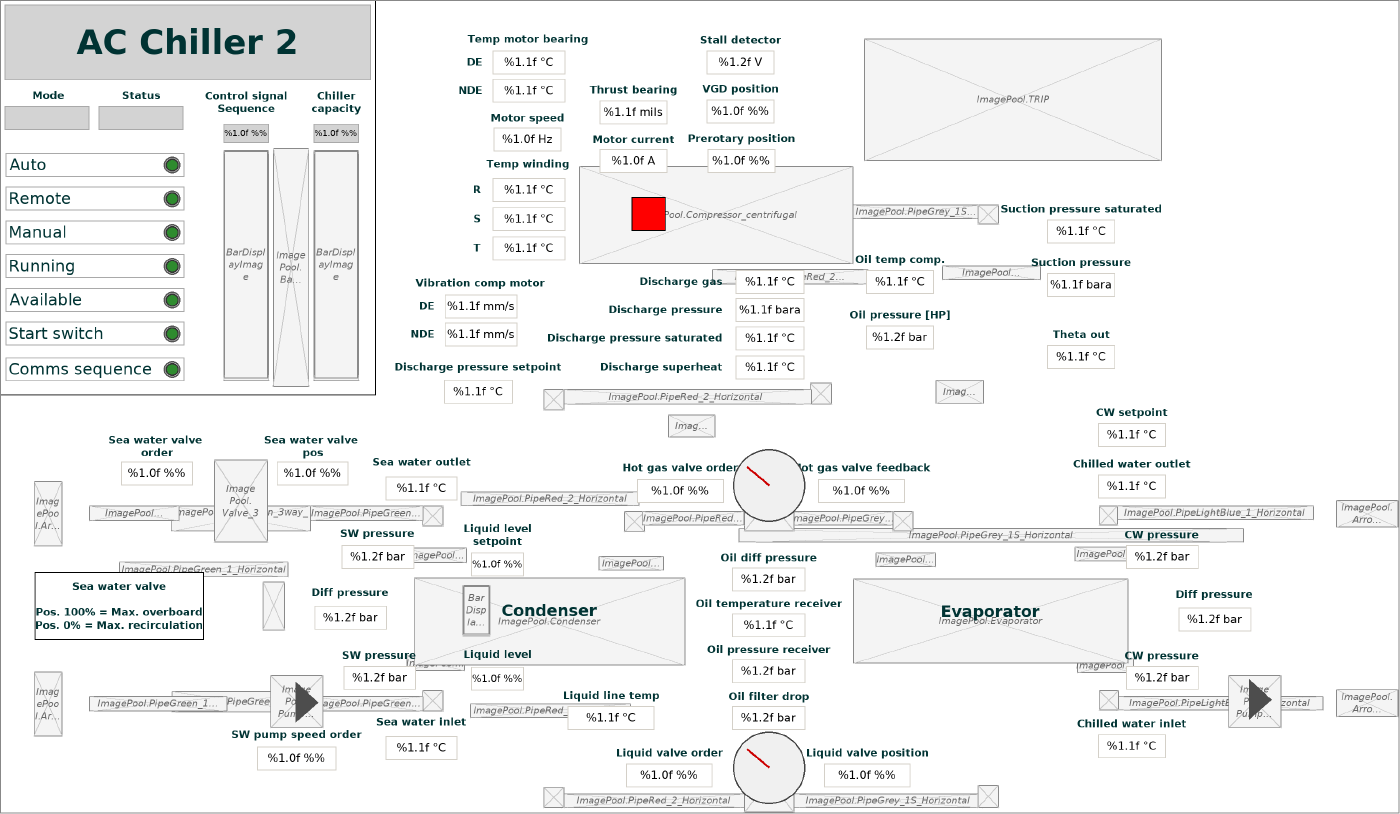
VISUALIZATION Chiller_2_Flow_Diagram  // 1492x868
    Rectangle (0,0 400x421)
    Textfield (238,132 48x20), "%1.0f %%", text variable: Sequence.Seq_cap_order_C1
        p4168582468: Sequence.Seq_cap_order_C1
    Image (1148,702 60x15), angle 270, image: ImagePool.PipeLightBlue_1_Horizontal
    Image (1145,583 67x15), angle 270, image: ImagePool.PipeLightBlue_1_Horizontal
    Image (908,218 137x15), image: ImagePool.PipeGrey_1S_Horizontal
    Image (845,846 202x15), image: ImagePool.PipeGrey_1S_Horizontal
    Image (933,589 64x15), angle 270, image: ImagePool.PipeGrey_1S_Horizontal
    Image (787,563 538x15), angle 270, image: ImagePool.PipeGrey_1S_Horizontal
    Image (843,545 110x15), image: ImagePool.PipeGrey_1S_Horizontal
    Image (638,593 69x15), angle 270, image: ImagePool.PipeRed_2_Horizontal
    Image (501,750 171x15), angle 270, image: ImagePool.PipeRed_2_Horizontal
    Label (218,94 89x30), "Control signal Sequence"
    Image (617,177 292x104), image: ImagePool.Compressor_centrifugal
    Image (759,287 166x16), angle 270, image: ImagePool.PipeRed_2_Horizontal
    Image (863,408 23x23), image: ImagePool.PipeRed_2_LU
    Image (596,415 269x16), image: ImagePool.PipeRed_2_Horizontal
    Image (909,617 293x90), image: ImagePool.Evaporator
    Image (431,584 66x16), angle 270, image: ImagePool.PipeGreen_1_Horizontal
    Image (450,539 22x22), image: ImagePool.PipeGreen_1_LD
    Image (329,539 122x16), image: ImagePool.PipeGreen_1_Horizontal
    Label (331,617 84x30), "Diff pressure"
    Textfield (335,646 77x25), "%1.2f bar", text variable: Chiller_2.dP_SW
        p4168582468: Chiller_2.dP_SW
    Image (127,599 180x16), angle 270, image: ImagePool.PipeGreen_1_Horizontal
    Image (183,737 147x22), image: ImagePool.PipeGreen_3way
    Image (433,699 62x16), angle 270, image: ImagePool.PipeGreen_1_Horizontal
    Image (450,736 22x22), image: ImagePool.PipeGreen_2_LU
    Image (329,742 122x16), image: ImagePool.PipeGreen_1_Horizontal
    Image (182,539 149x27), image: ImagePool.PipeGreen_3way_2
    Image (288,720 56x56), image: ImagePool.Pump_Large_3
    Polygon (315,746) (315,727) (339,749) (315,770) (315,762), colour toggle: Chiller_2.Sea_water_pump
    Image (36,513 30x69), angle 90, image: ImagePool.Arrow green down
    Image (36,716 30x69), angle 270, image: ImagePool.Arrow green down
    Image (579,415 22x22), image: ImagePool.PipeRed_1_RD
    Image (491,524 190x15), angle 270, image: ImagePool.PipeRed_2_Horizontal
    Label (360,554 84x30), "SW pressure"
    Textfield (364,581 77x25), "%1.2f bar", text variable: Chiller_2.Press_water_cond_out
        p4168582468: Chiller_2.Press_water_cond_out
    Image (95,539 96x16), image: ImagePool.PipeGreen_1_Horizontal
    Image (441,616 289x93), image: ImagePool.Condenser
    Image (598,846 197x15), image: ImagePool.PipeRed_2_Horizontal
    Image (579,839 22x22), image: ImagePool.PipeRed_2_RU
    Label (362,684 84x30), "SW pressure"
    Textfield (366,710 77x25), "%1.2f bar", text variable: Chiller_2.Press_water_cond_inlet
        p4168582468: Chiller_2.Press_water_cond_inlet
    Image (793,501 53x65), image: ImagePool.Valve_2
    Image (793,801 53x65), image: ImagePool.Valve_2
    Image (665,545 22x22), image: ImagePool.PipeRed_1_RD
    Image (684,545 109x15), image: ImagePool.PipeRed_2_Horizontal
    Image (951,545 22x21), image: ImagePool.PipeGrey_2_LD
    Image (1042,837 22x24), image: ImagePool.PipeGrey_3_LU
    Image (1042,218 22x21), image: ImagePool.PipeGrey_2_LD
    Image (1004,283 105x15), angle 270, image: ImagePool.PipeGrey_1S_Horizontal
    Label (521,636 129x30), "Condenser"
    Label (991,637 129x30), "Evaporator"
    Image (1189,539 211x15), image: ImagePool.PipeLightBlue_1_Horizontal
    Image (1171,539 20x21), image: ImagePool.PipeLightBlue_3_RD
    Image (1190,742 220x15), image: ImagePool.PipeLightBlue_1_Horizontal
    Image (1171,736 21x21), image: ImagePool.PipeLightBlue_3_RU
    Image (1424,533 66x29), angle 180, image: ImagePool.Arrow lightblue left
    Image (1424,735 66x29), image: ImagePool.Arrow lightblue left
    Image (1309,720 56x56), image: ImagePool.Pump_Large_3
    Polygon (1331,743) (1331,724) (1355,746) (1331,767) (1331,759), colour toggle: Chiller_2.CW_Flow_ind
    Image (280,620 23x52), image: ImagePool.Arrow green down
    Image (712,442 50x24), image: ImagePool.Arrow red left
    Image (997,405 51x25), angle 90, image: ImagePool.Arrow gray left
    Image (291,158 38x254), image: ImagePool.BarScale3
    Label (324,94 69x30), "Chiller capacity"
    Textfield (105,113 90x25), text list: 'TextList_PT', text index: Chiller_2.Unit_switch_status
    Textfield (5,113 90x25), text list: 'TextList_PT', text index: Chiller_2.Unit_start_switch
    Textfield (334,132 48x20), "%1.0f %%", text variable: Chiller_2.Chiller_capacity_t1
        p4168582468: Chiller_2.Chiller_capacity_t1
    Textfield (5,5 390x80), "AC Chiller 2"
    Label (521,160 84x30), "Temp winding"
    Textfield (525,190 77x25), "%1.1f °C", text variable: Chiller_2.Temp_motor_wind_R
        p4168582468: Chiller_2.Temp_motor_wind_R
    Label (496,190 25x25), "R"
    Textfield (525,221 77x25), "%1.1f °C", text variable: Chiller_2.Temp_motor_wind_S
        p4168582468: Chiller_2.Temp_motor_wind_S
    Label (496,221 25x25), "S"
    Textfield (525,252 77x25), "%1.1f °C", text variable: Chiller_2.Temp_motor_wind_T
        p4168582468: Chiller_2.Temp_motor_wind_T
    Label (496,252 25x25), "T"
    Textfield (679,511 92x25), "%1.0f %%", text variable: Chiller_2.Hot_gas_valve_output
        p4168582468: Chiller_2.Hot_gas_valve_output
    Label (664,484 122x30), "Hot gas valve order"
    Label (849,484 139x30), "Hot gas valve feedback"
    Textfield (872,511 92x25), "%1.0f %%", text variable: Chiller_2.Feedback_HGV
        p4168582468: Chiller_2.Feedback_HGV
    Meter360 (781,479 77x77), value: Chiller_2.Feedback_HGV, style: Meter-Meter360-Gray, scale format: %1.0f, scale 0..100
        p3451962224: ImagePool.Invisible
    Meter360 (781,780 77x77), value: Chiller_2.Feedback_liquid_valve, style: Meter-Meter360-Gray, scale format: %1.0f, scale 0..100
        p3451962224: ImagePool.Invisible
    Textfield (502,589 56x25), "%1.0f %%", text variable: Chiller_2.SP_PID_Level
        p4168582468: Chiller_2.SP_PID_Level
    Label (494,551 73x39), "Liquid level setpoint"
    Textfield (502,711 56x25), "%1.0f %%", text variable: Chiller_2.Liquid_level_condenser
        p4168582468: Chiller_2.Liquid_level_condenser
    Label (491,683 79x30), "Liquid level"
    Textfield (639,159 72x25), "%1.0f A", text variable: Chiller_2.Motor_current
        p4168582468: Chiller_2.Motor_current
    Label (634,138 83x22), "Motor current"
    Textfield (274,796 84x25), "%1.0f %%", text variable: Chiller_2.SW_pump_speed_order
        p4168582468: Chiller_2.SW_pump_speed_order
    Label (250,770 132x27), "SW pump speed order"
    Textfield (473,405 73x25), "%1.1f °C", tooltip "Chiller_2.SP_PID_seawater", text variable: Chiller_2.SP_PID_seawater
    Textfield (784,348 73x25), "%1.1f °C", text variable: Chiller_2.Discharge_saturated_temp
        p4168582468: Chiller_2.Discharge_saturated_temp
    Label (589,347 184x27), "Discharge pressure saturated"
    Label (425,378 169x27), "Discharge pressure setpoint"
    Textfield (411,785 76x25), "%1.1f °C", text variable: Chiller_2.Temp_water_inlet_cond
        p4168582468: Chiller_2.Temp_water_inlet_cond
    Label (399,755 100x30), "Sea water inlet"
    Textfield (411,508 76x25), "%1.1f °C", text variable: Chiller_2.Temp_water_outlet_cond
        p4168582468: Chiller_2.Temp_water_outlet_cond
    Label (397,478 105x30), "Sea water outlet"
    Label (500,27 126x30), "Temp motor bearing"
    Textfield (525,84 77x25), "%1.1f °C", text variable: Chiller_2.Temp_motor_bearing_NDE
        p4168582468: Chiller_2.Temp_motor_bearing_NDE
    Textfield (525,54 77x25), "%1.1f °C", text variable: Chiller_2.Temp_motor_bearing_DE
        p4168582468: Chiller_2.Temp_motor_bearing_DE
    Label (480,54 37x25), "DE"
    Label (480,84 37x25), "NDE"
    Label (678,287 95x27), "Discharge gas"
    Textfield (784,288 73x25), "%1.1f °C", text variable: Chiller_2.Temp_discharge
        p4168582468: Chiller_2.Temp_discharge
    Label (644,317 129x27), "Discharge pressure"
    Textfield (784,318 73x25), "%1.1f bara", text variable: Chiller_2.Press_discharge_compr
        p4168582468: Chiller_2.Press_discharge_compr
    Textfield (784,379 73x25), "%1.1f °C", text variable: Chiller_2.Discharge_superheat
        p4168582468: Chiller_2.Discharge_superheat
    Label (589,378 184x27), "Discharge superheat"
    Label (631,84 89x24), "Thrust bearing"
    Textfield (639,107 72x25), "%1.1f mils", text variable: Chiller_2.Thrust_bearing_position
        p4168582468: Chiller_2.Thrust_bearing_position
    Label (857,788 135x30), "Liquid valve position"
    Textfield (878,814 92x25), "%1.0f %%", text variable: Chiller_2.Feedback_liquid_valve
        p4168582468: Chiller_2.Feedback_liquid_valve
    Textfield (780,753 78x25), "%1.2f bar", text variable: Chiller_2.Oil_Filter_Drop
        p4168582468: Chiller_2.Oil_Filter_Drop
    Label (778,732 83x22), "Oil filter drop"
    Textfield (667,814 92x25), "%1.0f %%", text variable: Chiller_2.Liquid_valve_output
        p4168582468: Chiller_2.Liquid_valve_output
    Label (646,788 135x30), "Liquid valve order"
    Textfield (780,703 78x25), "%1.2f bar", text variable: Chiller_2.Press_oil_receiver
        p4168582468: Chiller_2.Press_oil_receiver
    Label (752,682 135x22), "Oil pressure receiver"
    Textfield (780,654 78x25), "%1.1f °C", text variable: Chiller_2.Oil_temp_receiver
        p4168582468: Chiller_2.Oil_temp_receiver
    Label (748,633 143x22), "Oil temperature receiver"
    Textfield (780,605 78x25), "%1.2f bar", text variable: Chiller_2.Oil_diff_pressure
        p4168582468: Chiller_2.Oil_diff_pressure
    Label (769,584 101x22), "Oil diff pressure"
    Label (738,136 105x24), "Prerotary position"
    Textfield (754,159 72x25), "%1.0f %%", text variable: Chiller_2.Feedback_PRV
        p4168582468: Chiller_2.Feedback_PRV
    Label (746,83 87x24), "VGD position"
    Textfield (753,106 72x25), "%1.0f %%", text variable: Chiller_2.Feedback_VGD
        p4168582468: Chiller_2.Feedback_VGD
    Label (746,31 87x24), "Stall detector"
    Textfield (753,54 72x25), "%1.2f V", text variable: Chiller_2.Stall_detector
        p4168582468: Chiller_2.Stall_detector
    Label (1067,211 171x24), "Suction pressure saturated"
    Textfield (1116,234 72x25), "%1.1f °C", text variable: Chiller_2.Suction_saturated_temp
        p4168582468: Chiller_2.Suction_saturated_temp
    Textfield (1116,291 72x25), "%1.1f bara", text variable: Chiller_2.Press_suction_compr
        p4168582468: Chiller_2.Press_suction_compr
    Label (1067,268 171x24), "Suction pressure"
    Textfield (1116,368 72x25), "%1.1f °C", text variable: Chiller_2.Theta_out
        p4168582468: Chiller_2.Theta_out
    Label (1111,345 83x24), "Theta out"
    Label (1196,557 84x27), "CW pressure"
    Textfield (1200,581 77x25), "%1.2f bar", text variable: Chiller_2.Press_chilled_medium_out
        p4168582468: Chiller_2.Press_chilled_medium_out
    Textfield (1200,710 77x25), "%1.2f bar", text variable: Chiller_2.Press_chilled_medium_in
        p4168582468: Chiller_2.Press_chilled_medium_in
    Label (1196,686 84x27), "CW pressure"
    Textfield (1170,506 72x25), "%1.1f °C", text variable: Chiller_2.Temp_chilled_medium_out
        p4168582468: Chiller_2.Temp_chilled_medium_out
    Label (1146,483 121x24), "Chilled water outlet"
    Label (1146,428 121x24), "CW setpoint"
    Textfield (1170,451 72x25), "%1.1f °C", text variable: Chiller_2.SP_CW_controller
        p4168582468: Chiller_2.SP_CW_controller
    Label (1252,619 84x30), "Diff pressure"
    Textfield (1256,648 77x25), "%1.2f bar", text variable: Chiller_2.dP_CW
        p4168582468: Chiller_2.dP_CW
    Textfield (1170,783 72x25), "%1.1f °C", text variable: Chiller_2.Temp_chilled_medium_in
        p4168582468: Chiller_2.Temp_chilled_medium_in
    Label (1146,760 121x24), "Chilled water inlet"
    Group (6,271 190x25)
        Rectangle (0,0 190x25)
        Label (0,2 105x21), "Running"
        Lamp1 (166,3 23x20), variable: Chiller_2.Unit_running, style: Lamp-Lamp1-Green
    Group (6,163 190x25)
        Rectangle (0,0 190x25)
        Label (1,2 105x21), "Auto"
        Lamp1 (166,3 23x20), variable: Chiller_2.Unit_auto, style: Lamp-Lamp1-Green
    Group (6,199 190x25)
        Rectangle (0,0 190x25)
        Label (0,2 105x21), "Remote"
        Lamp1 (166,3 23x20), variable: Chiller_2.Unit_remote, style: Lamp-Lamp1-Green
    Group (6,235 190x25)
        Rectangle (0,0 190x25)
        Label (0,2 105x21), "Manual"
        Lamp1 (166,3 23x20), variable: Chiller_2.Unit_manual, style: Lamp-Lamp1-Green
    Group (6,307 190x25)
        Rectangle (0,0 190x25)
        Label (1,2 105x21), "Available"
        Lamp1 (166,3 23x20), variable: Chiller_2.Unit_available, style: Lamp-Lamp1-Green
    Group (6,343 190x25)
        Rectangle (0,0 190x25)
        Label (0,2 130x21), "Start switch"
        Lamp1 (166,3 23x20), variable: Chiller_2.Unit_start_switch, style: Lamp-Lamp1-Green
    Group (6,381 190x25)
        Rectangle (0,0 190x25)
        Label (0,2 160x21), "Comms sequence"
        Lamp1 (166,3 23x20), variable: not.Sequence.A_Comms_chiller_1, style: Lamp-Lamp1-Green
    Label (912,265 95x24), "Oil temp comp."
    Textfield (923,288 72x25), "%1.1f °C", text variable: Chiller_2.Temp_oil_inlet_compr
        p4168582468: Chiller_2.Temp_oil_inlet_compr
    Label (902,324 115x24), "Oil pressure [HP]"
    Textfield (923,347 72x25), "%1.2f bar", text variable: Chiller_2.Press_oil_compr
        p4168582468: Chiller_2.Press_oil_compr
    Image (921,41 317x130), invisible if: Chiller_2.Unit_alarm, image: ImagePool.ALARM
    Image (921,41 317x130), invisible if: Chiller_2.Unit_trip, image: ImagePool.TRIP
    Label (7,87 89x30), "Mode"
    Label (106,87 89x30), "Status"
    Rectangle (334,160 48x246)
    Image (238,160 48x246), image: ImagePool.CapBarTranparant
    BarDisplayImage (239,161 46x242), value: Sequence.Seq_cap_order_C1, style: BarDisplayImage-Gray, scale format: %.0f, scale 0..100
        p3451962224: ImagePool.Invisible
    Rectangle (673,210 36x36), colour toggle: Chiller_2.Unit_running
    Rectangle (673,210 36x36), colour toggle: Chiller_2.Unit_alarm
    Rectangle (673,210 36x36), colour toggle: Chiller_2.Unit_trip
    Image (334,160 48x246), image: ImagePool.CapBarTranparant
    BarDisplayImage (335,161 46x242), value: Chiller_2.Chiller_capacity_t1, style: BarDisplayImage-Gray, scale format: %.0f, scale 0..100
        p3451962224: ImagePool.Invisible
    Rectangle (493,624 28x52)
    Image (493,624 29x54), image: ImagePool.CapBarTranparant
    BarDisplayImage (494,625 27x51), value: Chiller_2.Liquid_level_condenser, style: BarDisplayImage-Gray, scale format: %.0f, scale 0..100
        p3451962224: ImagePool.Invisible
    Image (95,742 147x16), image: ImagePool.PipeGreen_1_Horizontal
    Textfield (605,753 92x25), "%1.1f °C", text variable: Chiller_2.Liquid_line_temp
        p4168582468: Chiller_2.Liquid_line_temp
    Label (595,727 113x30), "Liquid line temp"
    Label (435,287 154x30), "Vibration comp motor"
    Textfield (474,344 77x25), "%1.1f mm/s", text variable: Chiller_2.Vibration_compressor_NDE
        p4168582468: Chiller_2.Vibration_compressor_NDE
    Textfield (474,314 77x25), "%1.1f mm/s", text variable: Chiller_2.Vibration_compressor_DE
        p4168582468: Chiller_2.Vibration_compressor_DE
    Label (429,314 37x25), "DE"
    Label (429,344 37x25), "NDE"
    Image (228,490 57x88), image: ImagePool.Valve_3
    Label (115,461 105x30), "Sea water valve order"
    Textfield (129,492 76x25), "%1.0f %%", text variable: Chiller_2.Control_signal_SW_valve
        p4168582468: Chiller_2.Control_signal_SW_valve
    Label (281,461 105x30), "Sea water valve pos"
    Textfield (295,492 76x25), "%1.0f %%", text variable: Chiller_2.Feedback_sea_water_valve
        p4168582468: Chiller_2.Feedback_sea_water_valve
    Group (37,610 180x72)
        Rectangle (0,0 180x72)
        Label (0,0 180x72), "Sea water valve Pos. 100% = Max. overboard Pos. 0% = Max. recirculation"
    Label (521,115 83x22), "Motor speed"
    Textfield (526,136 72x25), "%1.0f Hz", text variable: Chiller_2.Opt_speed_VFD_Hz
        p4168582468: Chiller_2.Opt_speed_VFD_Hz
END_VISUALIZATION

// /Chiller_2_Oil
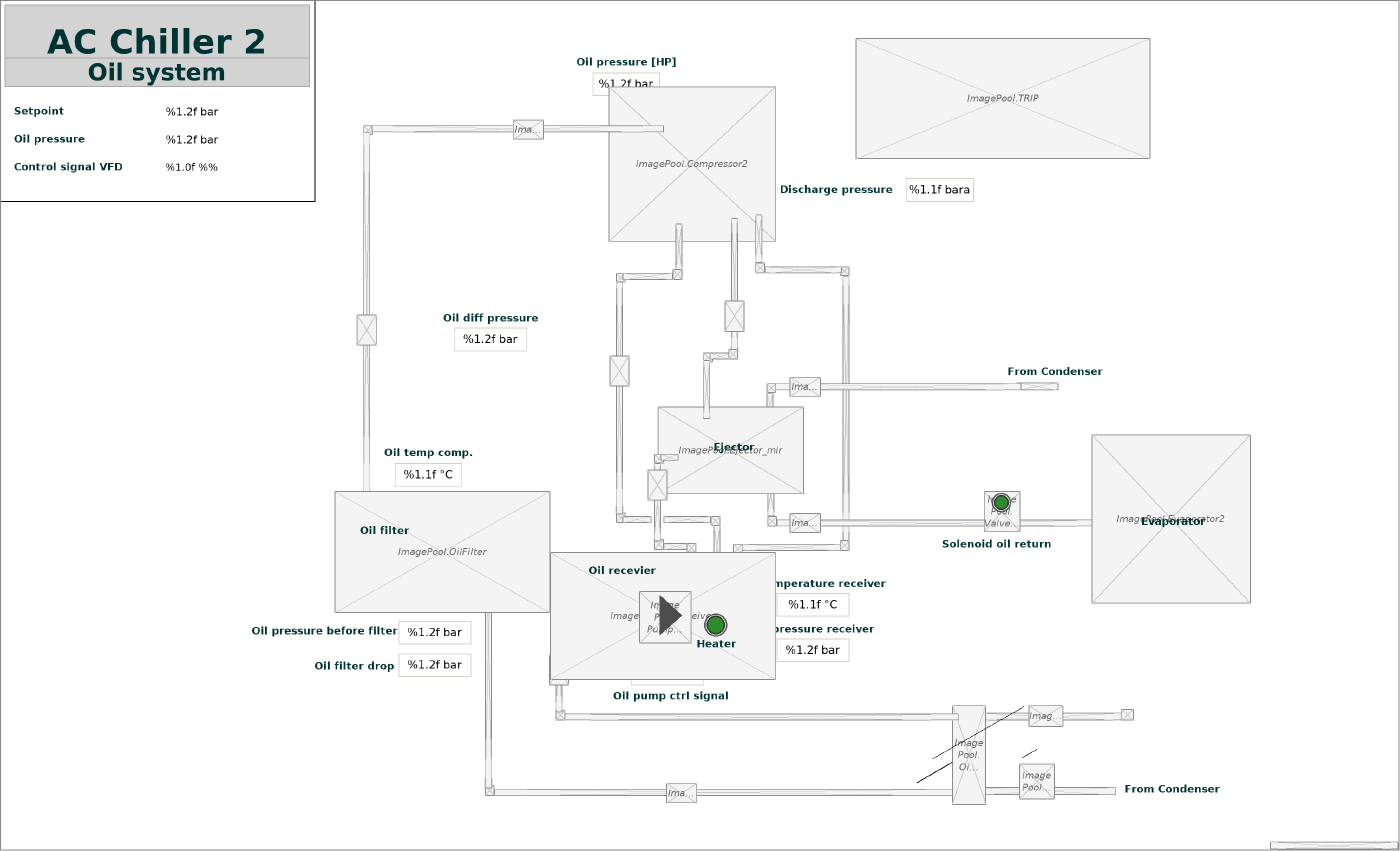
VISUALIZATION Chiller_2_Oil  // 1507x917
    Image (1094,412 45x8), angle 180, image: ImagePool.PipeBlack_1S_H_Faded
    Rectangle (0,0 339x217)
    Image (1367,907 138x8), angle 270, image: ImagePool.PipeGrey_1S_Horizontal
    Image (1053,768 155x8), image: ImagePool.PipeGrey_1S_Horizontal
    Image (1207,764 13x12), image: ImagePool.PipeGrey_3_LU
    Textfield (5,5 328x80), "AC Chiller 2"
    Label (1093,387 97x27), "From Condenser"
    Label (835,191 129x27), "Discharge pressure"
    Textfield (975,192 73x25), "%1.1f bara", text variable: Chiller_2.Press_discharge_compr
        p4168582468: Chiller_2.Press_discharge_compr
    Label (1029,573 106x27), "Solenoid oil return"
    Textfield (429,704 78x25), "%1.2f bar", text variable: Chiller_2.Oil_Filter_Drop
        p4168582468: Chiller_2.Oil_Filter_Drop
    Label (340,707 83x22), "Oil filter drop"
    Textfield (836,688 78x25), "%1.2f bar", text variable: Chiller_2.Press_oil_receiver
        p4168582468: Chiller_2.Press_oil_receiver
    Label (808,667 135x22), "Oil pressure receiver"
    Textfield (836,639 78x25), "%1.1f °C", text variable: Chiller_2.Oil_temp_receiver
        p4168582468: Chiller_2.Oil_temp_receiver
    Label (804,618 143x22), "Oil temperature receiver"
    Textfield (489,353 78x25), "%1.2f bar", text variable: Chiller_2.Oil_diff_pressure
        p4168582468: Chiller_2.Oil_diff_pressure
    Label (478,332 101x22), "Oil diff pressure"
    Label (414,476 95x24), "Oil temp comp."
    Textfield (425,499 72x25), "%1.1f °C", text variable: Chiller_2.Temp_oil_inlet_compr
        p4168582468: Chiller_2.Temp_oil_inlet_compr
    Label (617,55 115x24), "Oil pressure [HP]"
    Textfield (638,78 72x25), "%1.2f bar", text variable: Chiller_2.Press_oil_compr
        p4168582468: Chiller_2.Press_oil_compr
    Image (921,41 317x130), invisible if: not.Chiller_2.Unit_alarm, image: ImagePool.ALARM
    Image (921,41 317x130), invisible if: not.Chiller_2.Unit_trip, image: ImagePool.TRIP
    Textfield (5,62 328x31), "Oil system"
    Textfield (178,109 57x23), "%1.2f bar", tooltip "Chiller_2.SP_oil_pressure_diff", text variable: Chiller_2.SP_oil_pressure_diff
    Label (12,105 106x30), "Setpoint"
    Textfield (178,139 57x23), "%1.2f bar", tooltip "Chiller_2.Oil_diff_pressure", text variable: Chiller_2.Oil_diff_pressure
    Label (12,135 107x30), "Oil pressure"
    Textfield (178,169 57x23), "%1.0f %%", tooltip "Chiller_2.SP_freq_oil_pump_VFD", text variable: Chiller_2.SP_freq_oil_pump_VFD
    Label (12,165 109x30), "Control signal VFD"
    Textfield (679,713 78x25), "%1.2f Hz", tooltip "Chiller_2.SP_freq_oil_pump_VFD", text variable: Chiller_2.Press_oil_receiver
    Label (655,739 135x22), "Oil pump ctrl signal"
    Textfield (429,669 78x25), "%1.2f bar", text variable: Chiller_2.Oil_pressure_before_filter
        p4168582468: Chiller_2.Oil_pressure_before_filter
    Label (276,669 147x22), "Oil pressure before filter"
    Label (1210,837 106x27), "From Condenser"
    Image (655,93 180x167), image: ImagePool.Compressor2
    Image (1051,848 150x8), angle 180, image: ImagePool.PipeBlack_1S_H_Faded
    Image (798,586 108x7), image: ImagePool.PipeBlack_1_Horizontal
    Image (907,297 7x286), image: ImagePool.PipeBlack_1_Vertical
    Image (391,135 10x10), image: ImagePool.PipeBlack_1_RD
    Image (522,846 10x11), image: ImagePool.PipeBlack_1_RU
    Image (1107,760 37x23), image: ImagePool.Arrow gray right
    Image (836,560 348x7), image: ImagePool.PipeBlack_1_Horizontal
    Image (1175,468 171x182), image: ImagePool.Evaporator2
    Image (826,512 7x44), image: ImagePool.PipeBlack_1_Vertical
    Image (826,556 10x11), image: ImagePool.PipeBlack_1_RU
    Image (789,596 7x28), image: ImagePool.PipeBlack_1_Vertical
    Image (789,586 10x10), image: ImagePool.PipeBlack_1_RD
    Image (904,582 10x11), image: ImagePool.PipeBlack_1_LU
    Image (850,553 33x21), image: ImagePool.Arrow black left
    Image (904,287 10x10), image: ImagePool.PipeBlack_1_LD
    Image (823,287 83x7), image: ImagePool.PipeBlack_1_Horizontal
    Image (813,283 10x11), image: ImagePool.PipeBlack_1_RU
    Image (813,231 7x52), image: ImagePool.PipeBlack_1_Vertical
    Image (825,413 10x10), image: ImagePool.PipeBlack_1_RD
    Image (834,413 265x7), image: ImagePool.PipeBlack_1_Horizontal
    Image (825,423 7x28), image: ImagePool.PipeBlack_1_Vertical
    Image (708,438 157x94), image: ImagePool.Ejector_mir
    Image (850,406 33x21), image: ImagePool.Arrow black left
    Image (532,850 500x7), image: ImagePool.PipeBlack_1_Horizontal
    Image (1025,760 36x107), image: ImagePool.OilHeatExchanger
    Image (605,769 427x7), image: ImagePool.PipeBlack_1_Horizontal
    Image (598,765 10x11), image: ImagePool.PipeBlack_1_RU
    Image (598,670 7x97), image: ImagePool.PipeBlack_1_Vertical
    Image (598,660 10x10), image: ImagePool.PipeBlack_1_RD
    Image (605,660 19x7), image: ImagePool.PipeBlack_1_Horizontal
    Image (591,705 21x33), image: ImagePool.Arrow black down
    Image (717,844 33x21), image: ImagePool.Arrow black left
    Image (768,566 7x50), image: ImagePool.PipeBlack_1_Vertical
    Image (765,556 10x10), image: ImagePool.PipeBlack_1_LD
    Image (714,556 51x7), image: ImagePool.PipeBlack_1_Horizontal
    Image (704,581 10x11), image: ImagePool.PipeBlack_1_RU
    Image (704,499 7x84), image: ImagePool.PipeBlack_1_Vertical
    Image (704,489 10x10), image: ImagePool.PipeBlack_1_RD
    Image (711,489 19x7), image: ImagePool.PipeBlack_1_Horizontal
    Image (697,506 21x33), image: ImagePool.Arrow black down
    Image (714,585 28x7), image: ImagePool.PipeBlack_1_Horizontal
    Image (739,585 10x10), image: ImagePool.PipeBlack_1_LD
    Image (742,595 7x21), image: ImagePool.PipeBlack_1_Vertical
    Image (592,595 243x137), image: ImagePool.OilReceiver
    Image (400,135 314x7), image: ImagePool.PipeBlack_1_Horizontal
    Label (630,604 80x22), "Oil recevier"
    Image (522,553 7x296), image: ImagePool.PipeBlack_1_Vertical
    Image (519,544 10x10), image: ImagePool.PipeBlack_1_LD
    Image (400,544 120x7), image: ImagePool.PipeBlack_1_Horizontal
    Image (391,540 10x11), image: ImagePool.PipeBlack_1_RU
    Image (391,142 7x400), image: ImagePool.PipeBlack_1_Vertical
    Image (663,552 10x11), image: ImagePool.PipeBlack_1_RU
    Image (663,301 7x253), image: ImagePool.PipeBlack_1_Vertical
    Image (663,294 10x10), image: ImagePool.PipeBlack_1_RD
    Image (670,294 54x7), image: ImagePool.PipeBlack_1_Horizontal
    Image (656,383 21x33), image: ImagePool.Arrow black down
    Image (670,556 31x7), image: ImagePool.PipeBlack_1_Horizontal
    Image (727,241 7x53), image: ImagePool.PipeBlack_1_Vertical
    Image (724,290 10x11), image: ImagePool.PipeBlack_1_LU
    Image (757,380 10x10), image: ImagePool.PipeBlack_1_RD
    Image (764,380 22x7), image: ImagePool.PipeBlack_1_Horizontal
    Image (787,235 7x144), image: ImagePool.PipeBlack_1_Vertical
    Image (784,376 10x11), image: ImagePool.PipeBlack_1_LU
    Image (757,388 7x63), image: ImagePool.PipeBlack_1_Vertical
    Image (780,324 21x33), image: ImagePool.Arrow black down
    Label (750,471 80x22), "Ejector"
    Label (1223,551 80x22), "Evaporator"
    Image (384,339 21x33), image: ImagePool.Arrow black up
    Image (552,129 33x21), image: ImagePool.Arrow black right
    Image (360,529 232x131), image: ImagePool.OilFilter
    Label (387,561 54x22), "Oil filter"
    Line (987,843) (1025,821)
    Line (1100,816) (1116,807)
    Line (1004,817) (1102,761)
    Image (1097,823 38x38), image: ImagePool.RegValve
    Image (688,637 56x56), image: ImagePool.Pump_Large_3
    Polygon (710,660) (710,641) (734,663) (710,684) (710,676), colour toggle: Chiller_2.Comp_oil_pump
    Lamp1 (756,656 29x35), variable: Chiller_2.Oil_heater, style: Lamp-Lamp1-Green
    Label (744,683 55x22), "Heater"
    Image (1059,529 39x44), image: ImagePool.Valve_2
    Lamp1 (1066,529 24x25), variable: Chiller_2.Solenoid_oil_return, style: Lamp-Lamp1-Green
END_VISUALIZATION

